KUKA KRL program: f1_Kuka_APT225T02S25.SRC

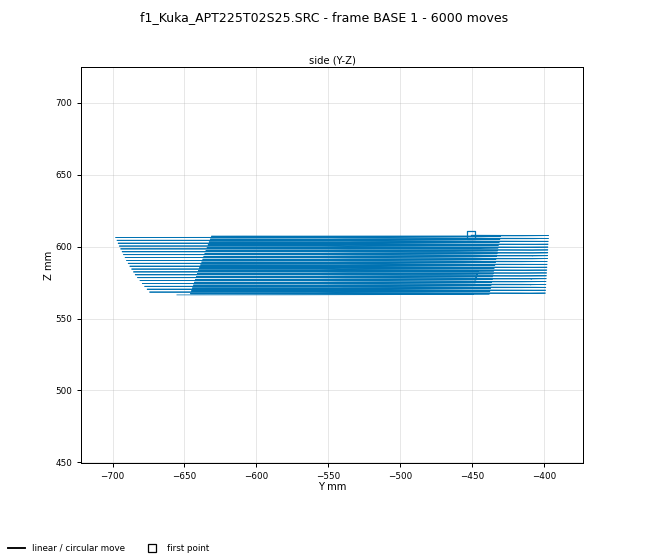
[picture p0: tool path of f1_Kuka_APT225T02S25.SRC in frame BASE 1, 6000 of 6001 moves have a stored position in this frame; points joined in program order, loops and branches not executed]
&ACCESS RVP
&REL 2
&PARAM TEMPLATE = C:\KRC\Roboter\Template\vorgabe
&PARAM EDITMASK = *
DEF f1_Kuka_APT225T02S25()


;FOLD INI;%{PE}%V3.2.0,%MKUKATPBASIS,%CINIT,%VCOMMON,%P
  ;FOLD BAS INI;%{E}%V3.2.0,%MKUKATPBASIS,%CINIT,%VINIT,%P
    GLOBAL INTERRUPT DECL 3 WHEN $STOPMESS==TRUE DO IR_STOPM ( )
    INTERRUPT ON 3
    BAS (#INITMOV,0 )
  ;ENDFOLD (BAS INI)
  ;FOLD USER INI;%{E}%V3.2.0,%MKUKATPUSER,%CINIT,%VINIT,%P
    ;Make your modifications here
  ;ENDFOLD (USER INI)
;ENDFOLD (INI)


;*** Make Null PTP Move
  PTP $pos_act

;*** Auto Load The Correct TOOL Data
  $tool=tool_data[2]

;*** Auto Load The Correct BASE Data
  $base=base_data[1]

  $ADVANCE = 5

;*** Restate Last Velocity
MMPM(30000.0)
SetRPM(8000)
LIN {X -0.035,Y -450.597,Z 607.985,A 0.000,B 0.000,C 90.000,E1 213.214} C_DIS
LIN {X 0.136,Y -446.521,Z 607.972,A 0.000,B 0.000,C 90.000,E1 210.924} C_DIS
LIN {X -0.250,Y -442.434,Z 607.959,A 0.000,B 0.000,C 90.000,E1 208.693} C_DIS
LIN {X 0.124,Y -440.119,Z 607.952,A 0.000,B 0.000,C 90.000,E1 207.334} C_DIS
LIN {X -0.104,Y -437.231,Z 607.943,A 0.000,B 0.000,C 90.000,E1 205.720} C_DIS
LIN {X -0.186,Y -434.380,Z 607.934,A 0.000,B 0.000,C 90.000,E1 204.079} C_DIS
LIN {X 0.098,Y -430.481,Z 607.921,A 0.000,B 0.000,C 90.000,E1 201.716} C_DIS
LIN {X -0.046,Y -427.723,Z 607.911,A 0.000,B 0.000,C 90.000,E1 200.066} C_DIS
LIN {X 0.139,Y -423.997,Z 607.898,A 0.000,B 0.000,C 90.000,E1 197.692} C_DIS
LIN {X -0.165,Y -420.659,Z 607.885,A 0.000,B 0.000,C 90.000,E1 195.371} C_DIS
LIN {X -0.117,Y -418.759,Z 607.878,A 0.000,B 0.000,C 90.000,E1 194.008} C_DIS
LIN {X 0.000,Y -415.623,Z 607.866,A 0.000,B 0.000,C 90.000,E1 191.951} C_DIS
LIN {X 0.069,Y -411.377,Z 607.849,A 0.000,B 0.000,C 90.000,E1 188.859} C_DIS
LIN {X 0.166,Y -409.163,Z 607.840,A 0.000,B 0.000,C 90.000,E1 187.125} C_DIS
LIN {X 0.188,Y -406.047,Z 607.826,A 0.000,B 0.000,C 90.000,E1 184.702} C_DIS
LIN {X -0.104,Y -401.893,Z 607.805,A 0.000,B 0.000,C 90.000,E1 180.917} C_DIS
LIN {X 0.005,Y -399.883,Z 607.791,A 0.000,B 0.000,C 90.000,E1 178.453} C_DIS
LIN {X -0.042,Y -397.946,Z 607.772,A 0.000,B 0.000,C 90.000,E1 174.951} C_DIS
LIN {X 0.089,Y -397.239,Z 607.758,A 0.000,B 0.000,C 90.000,E1 172.470} C_DIS
LIN {X -0.143,Y -396.829,Z 607.745,A 0.000,B 0.000,C 90.000,E1 170.038} C_DIS
LIN {X 0.183,Y -396.837,Z 607.729,A 0.000,B 0.000,C 90.000,E1 167.173} C_DIS
LIN {X -0.078,Y -397.303,Z 607.713,A 0.000,B 0.000,C 90.000,E1 164.393} C_DIS
LIN {X 0.094,Y -397.670,Z 607.705,A 0.000,B 0.000,C 90.000,E1 162.960} C_DIS
LIN {X 0.110,Y -398.325,Z 607.692,A 0.000,B 0.000,C 90.000,E1 160.496} C_DIS
LIN {X -0.123,Y -398.904,Z 607.682,A 0.000,B 0.000,C 90.000,E1 158.773} C_DIS
LIN {X -0.113,Y -399.695,Z 607.670,A 0.000,B 0.000,C 90.000,E1 156.666} C_DIS
LIN {X 0.072,Y -400.529,Z 607.659,A 0.000,B 0.000,C 90.000,E1 154.537} C_DIS
LIN {X 0.076,Y -401.373,Z 607.647,A 0.000,B 0.000,C 90.000,E1 152.436} C_DIS
LIN {X -0.127,Y -402.008,Z 607.637,A 0.000,B 0.000,C 90.000,E1 150.717} C_DIS
LIN {X -0.068,Y -402.708,Z 607.626,A 0.000,B 0.000,C 90.000,E1 148.614} C_DIS
LIN {X 0.077,Y -403.311,Z 607.614,A 0.000,B 0.000,C 90.000,E1 146.501} C_DIS
LIN {X 0.131,Y -403.912,Z 607.602,A 0.000,B 0.000,C 90.000,E1 144.402} C_DIS
LIN {X 0.002,Y -404.655,Z 607.589,A 0.000,B 0.000,C 90.000,E1 141.984} C_DIS
LIN {X -0.068,Y -405.359,Z 607.577,A 0.000,B 0.000,C 90.000,E1 139.908} C_DIS
LIN {X 0.004,Y -405.810,Z 607.568,A 0.000,B 0.000,C 90.000,E1 138.162} C_DIS
LIN {X 0.028,Y -406.293,Z 607.554,A 0.000,B 0.000,C 90.000,E1 135.729} C_DIS
LIN {X 0.215,Y -406.624,Z 607.543,A 0.000,B 0.000,C 90.000,E1 133.623} C_DIS
LIN {X -0.133,Y -406.875,Z 607.535,A 0.000,B 0.000,C 90.000,E1 132.285} C_DIS
LIN {X 0.111,Y -407.271,Z 607.523,A 0.000,B 0.000,C 90.000,E1 130.172} C_DIS
LIN {X 0.085,Y -407.637,Z 607.515,A 0.000,B 0.000,C 90.000,E1 128.705} C_DIS
LIN {X 0.252,Y -415.304,Z 607.500,A 0.000,B 0.000,C 90.000,E1 126.011} C_DIS
LIN {X -0.037,Y -417.748,Z 607.495,A 0.000,B 0.000,C 90.000,E1 125.025} C_DIS
LIN {X 0.201,Y -421.789,Z 607.486,A 0.000,B 0.000,C 90.000,E1 123.372} C_DIS
LIN {X 0.162,Y -421.843,Z 607.486,A 0.000,B 0.000,C 90.000,E1 123.372} C_DIS
LIN {X 0.201,Y -422.819,Z 607.485,A 0.000,B 0.000,C 90.000,E1 123.293} C_DIS
LIN {X -0.069,Y -426.964,Z 607.484,A 0.000,B 0.000,C 90.000,E1 123.086} C_DIS
LIN {X -0.088,Y -450.936,Z 607.477,A 0.000,B 0.000,C 90.000,E1 121.878} C_DIS
LIN {X 0.091,Y -460.950,Z 607.474,A 0.000,B 0.000,C 90.000,E1 121.337} C_DIS
LIN {X 0.206,Y -472.469,Z 607.471,A 0.000,B 0.000,C 90.000,E1 120.669} C_DIS
LIN {X -0.047,Y -482.176,Z 607.467,A 0.000,B 0.000,C 90.000,E1 120.129} C_DIS
LIN {X -0.197,Y -488.571,Z 607.465,A 0.000,B 0.000,C 90.000,E1 119.745} C_DIS
LIN {X 0.182,Y -498.111,Z 607.462,A 0.000,B 0.000,C 90.000,E1 119.077} C_DIS
LIN {X -0.210,Y -504.249,Z 607.459,A 0.000,B 0.000,C 90.000,E1 118.693} C_DIS
LIN {X 0.009,Y -511.965,Z 607.456,A 0.000,B 0.000,C 90.000,E1 118.103} C_DIS
LIN {X 0.049,Y -518.096,Z 607.454,A 0.000,B 0.000,C 90.000,E1 117.641} C_DIS
LIN {X -0.222,Y -527.985,Z 607.449,A 0.000,B 0.000,C 90.000,E1 116.873} C_DIS
LIN {X 0.112,Y -533.671,Z 607.447,A 0.000,B 0.000,C 90.000,E1 116.360} C_DIS
LIN {X 0.246,Y -539.267,Z 607.444,A 0.000,B 0.000,C 90.000,E1 115.848} C_DIS
LIN {X -0.034,Y -544.196,Z 607.441,A 0.000,B 0.000,C 90.000,E1 115.412} C_DIS
LIN {X 0.283,Y -549.010,Z 607.439,A 0.000,B 0.000,C 90.000,E1 114.899} C_DIS
LIN {X 0.037,Y -553.759,Z 607.436,A 0.000,B 0.000,C 90.000,E1 114.387} C_DIS
LIN {X 0.105,Y -558.121,Z 607.432,A 0.000,B 0.000,C 90.000,E1 113.823} C_DIS
LIN {X 0.087,Y -562.823,Z 607.429,A 0.000,B 0.000,C 90.000,E1 113.131} C_DIS
LIN {X -0.203,Y -567.599,Z 607.424,A 0.000,B 0.000,C 90.000,E1 112.333} C_DIS
LIN {X 0.089,Y -571.862,Z 607.419,A 0.000,B 0.000,C 90.000,E1 111.482} C_DIS
LIN {X 0.188,Y -575.169,Z 607.416,A 0.000,B 0.000,C 90.000,E1 110.791} C_DIS
LIN {X 0.107,Y -578.237,Z 607.412,A 0.000,B 0.000,C 90.000,E1 110.120} C_DIS
LIN {X -0.031,Y -581.512,Z 607.407,A 0.000,B 0.000,C 90.000,E1 109.322} C_DIS
LIN {X 0.225,Y -584.590,Z 607.403,A 0.000,B 0.000,C 90.000,E1 108.489} C_DIS
LIN {X 0.144,Y -587.415,Z 607.398,A 0.000,B 0.000,C 90.000,E1 107.692} C_DIS
LIN {X 0.156,Y -590.709,Z 607.392,A 0.000,B 0.000,C 90.000,E1 106.622} C_DIS
LIN {X 0.221,Y -593.690,Z 607.387,A 0.000,B 0.000,C 90.000,E1 105.552} C_DIS
LIN {X 0.184,Y -600.514,Z 607.373,A 0.000,B 0.000,C 90.000,E1 103.175} C_DIS
LIN {X 0.275,Y -605.256,Z 607.365,A 0.000,B 0.000,C 90.000,E1 101.591} C_DIS
LIN {X 0.273,Y -608.432,Z 607.359,A 0.000,B 0.000,C 90.000,E1 100.546} C_DIS
LIN {X 0.064,Y -612.242,Z 607.352,A 0.000,B 0.000,C 90.000,E1 99.265} C_DIS
LIN {X -0.179,Y -615.776,Z 607.344,A 0.000,B 0.000,C 90.000,E1 97.992} C_DIS
LIN {X -0.041,Y -618.497,Z 607.339,A 0.000,B 0.000,C 90.000,E1 96.947} C_DIS
LIN {X 0.055,Y -621.080,Z 607.333,A 0.000,B 0.000,C 90.000,E1 95.910} C_DIS
LIN {X -0.119,Y -623.777,Z 607.326,A 0.000,B 0.000,C 90.000,E1 94.645} C_DIS
LIN {X -0.088,Y -624.817,Z 607.323,A 0.000,B 0.000,C 90.000,E1 94.131} C_DIS
LIN {X -0.203,Y -626.978,Z 607.316,A 0.000,B 0.000,C 90.000,E1 92.865} C_DIS
LIN {X -0.069,Y -628.522,Z 607.310,A 0.000,B 0.000,C 90.000,E1 91.835} C_DIS
LIN {X -0.162,Y -630.042,Z 607.303,A 0.000,B 0.000,C 90.000,E1 90.573} C_DIS
LIN {X -0.072,Y -630.506,Z 607.300,A 0.000,B 0.000,C 90.000,E1 90.057} C_DIS
LIN {X 0.118,Y -631.128,Z 607.295,A 0.000,B 0.000,C 90.000,E1 89.026} C_DIS
LIN {X -0.054,Y -631.303,Z 607.290,A 0.000,B 0.000,C 90.000,E1 88.282} C_DIS
LIN {X -0.112,Y -631.250,Z 607.283,A 0.000,B 0.000,C 90.000,E1 87.020} C_DIS
LIN {X 0.015,Y -631.105,Z 607.281,A 0.000,B 0.000,C 90.000,E1 86.502} C_DIS
LIN {X -0.050,Y -630.373,Z 607.274,A 0.000,B 0.000,C 90.000,E1 85.241} C_DIS
LIN {X 0.201,Y -629.528,Z 607.268,A 0.000,B 0.000,C 90.000,E1 84.204} C_DIS
LIN {X -0.180,Y -628.525,Z 607.262,A 0.000,B 0.000,C 90.000,E1 83.223} C_DIS
LIN {X 0.045,Y -627.114,Z 607.257,A 0.000,B 0.000,C 90.000,E1 82.186} C_DIS
LIN {X 0.123,Y -625.043,Z 607.250,A 0.000,B 0.000,C 90.000,E1 80.905} C_DIS
LIN {X -0.221,Y -623.038,Z 607.244,A 0.000,B 0.000,C 90.000,E1 79.916} C_DIS
LIN {X 0.020,Y -620.933,Z 607.238,A 0.000,B 0.000,C 90.000,E1 78.870} C_DIS
LIN {X 0.218,Y -618.647,Z 607.233,A 0.000,B 0.000,C 90.000,E1 77.825} C_DIS
LIN {X -0.094,Y -616.179,Z 607.227,A 0.000,B 0.000,C 90.000,E1 76.825} C_DIS
LIN {X 0.069,Y -612.828,Z 607.220,A 0.000,B 0.000,C 90.000,E1 75.519} C_DIS
LIN {X 0.181,Y -609.203,Z 607.212,A 0.000,B 0.000,C 90.000,E1 74.212} C_DIS
LIN {X -0.003,Y -606.832,Z 607.208,A 0.000,B 0.000,C 90.000,E1 73.449} C_DIS
LIN {X -0.045,Y -604.265,Z 607.204,A 0.000,B 0.000,C 90.000,E1 72.670} C_DIS
LIN {X 0.075,Y -601.395,Z 607.199,A 0.000,B 0.000,C 90.000,E1 71.873} C_DIS
LIN {X -0.312,Y -597.101,Z 607.194,A 0.000,B 0.000,C 90.000,E1 70.859} C_DIS
LIN {X -0.067,Y -591.722,Z 607.187,A 0.000,B 0.000,C 90.000,E1 69.645} C_DIS
LIN {X 0.203,Y -588.653,Z 607.183,A 0.000,B 0.000,C 90.000,E1 68.954} C_DIS
LIN {X 0.169,Y -584.506,Z 607.179,A 0.000,B 0.000,C 90.000,E1 68.156} C_DIS
LIN {X 0.158,Y -580.904,Z 607.175,A 0.000,B 0.000,C 90.000,E1 67.486} C_DIS
LIN {X 0.260,Y -575.959,Z 607.171,A 0.000,B 0.000,C 90.000,E1 66.666} C_DIS
LIN {X -0.279,Y -572.428,Z 607.168,A 0.000,B 0.000,C 90.000,E1 66.177} C_DIS
LIN {X -0.172,Y -567.537,Z 607.164,A 0.000,B 0.000,C 90.000,E1 65.485} C_DIS
LIN {X -0.018,Y -563.248,Z 607.161,A 0.000,B 0.000,C 90.000,E1 64.921} C_DIS
LIN {X 0.103,Y -558.628,Z 607.158,A 0.000,B 0.000,C 90.000,E1 64.357} C_DIS
LIN {X 0.007,Y -553.569,Z 607.155,A 0.000,B 0.000,C 90.000,E1 63.819} C_DIS
LIN {X 0.279,Y -547.976,Z 607.152,A 0.000,B 0.000,C 90.000,E1 63.256} C_DIS
LIN {X -0.135,Y -543.643,Z 607.150,A 0.000,B 0.000,C 90.000,E1 62.922} C_DIS
LIN {X -0.010,Y -539.017,Z 607.148,A 0.000,B 0.000,C 90.000,E1 62.564} C_DIS
LIN {X 0.105,Y -533.075,Z 607.145,A 0.000,B 0.000,C 90.000,E1 62.153} C_DIS
LIN {X -0.007,Y -526.442,Z 607.143,A 0.000,B 0.000,C 90.000,E1 61.769} C_DIS
LIN {X 0.051,Y -519.547,Z 607.141,A 0.000,B 0.000,C 90.000,E1 61.385} C_DIS
LIN {X 0.000,Y -512.850,Z 607.139,A 0.000,B 0.000,C 90.000,E1 61.051} C_DIS
LIN {X 0.227,Y -500.895,Z 607.136,A 0.000,B 0.000,C 90.000,E1 60.461} C_DIS
LIN {X -0.159,Y -485.528,Z 607.132,A 0.000,B 0.000,C 90.000,E1 59.793} C_DIS
LIN {X -0.080,Y -468.875,Z 607.128,A 0.000,B 0.000,C 90.000,E1 58.997} C_DIS
LIN {X -0.240,Y -446.443,Z 607.121,A 0.000,B 0.000,C 90.000,E1 57.867} C_DIS
LIN {X -0.043,Y -446.380,Z 607.121,A 0.000,B 0.000,C 90.000,E1 57.837} C_DIS
LIN {X -0.065,Y -443.942,Z 607.114,A 0.000,B 0.000,C 90.000,E1 56.501} C_DIS
LIN {X 0.223,Y -434.128,Z 607.090,A 0.000,B 0.000,C 90.000,E1 52.190} C_DIS
LIN {X 0.064,Y -431.651,Z 607.083,A 0.000,B 0.000,C 90.000,E1 50.884} C_DIS
LIN {X -0.013,Y -430.264,Z 607.080,A 0.000,B 0.000,C 90.000,E1 50.312} C_DIS
LIN {X 0.057,Y -431.003,Z 607.074,A 0.000,B 0.000,C 90.000,E1 49.218} C_DIS
LIN {X 0.055,Y -432.039,Z 607.064,A 0.000,B 0.000,C 90.000,E1 47.553} C_DIS
LIN {X -0.083,Y -433.331,Z 607.051,A 0.000,B 0.000,C 90.000,E1 45.243} C_DIS
LIN {X -0.124,Y -434.602,Z 607.040,A 0.000,B 0.000,C 90.000,E1 43.257} C_DIS
LIN {X -0.086,Y -435.484,Z 607.031,A 0.000,B 0.000,C 90.000,E1 41.595} C_DIS
LIN {X 0.055,Y -436.199,Z 607.024,A 0.000,B 0.000,C 90.000,E1 40.253} C_DIS
LIN {X 0.158,Y -437.105,Z 607.013,A 0.000,B 0.000,C 90.000,E1 38.257} C_DIS
LIN {X 0.055,Y -437.585,Z 607.005,A 0.000,B 0.000,C 90.000,E1 36.950} C_DIS
LIN {X 0.005,Y -438.149,Z 606.994,A 0.000,B 0.000,C 90.000,E1 34.978} C_DIS
LIN {X -0.017,Y -438.398,Z 606.989,A 0.000,B 0.000,C 90.000,E1 33.992} C_DIS
LIN {X -0.009,Y -438.614,Z 606.982,A 0.000,B 0.000,C 90.000,E1 32.673} C_DIS
LIN {X -0.131,Y -439.071,Z 606.969,A 0.000,B 0.000,C 90.000,E1 30.384} C_DIS
LIN {X 0.124,Y -439.584,Z 606.954,A 0.000,B 0.000,C 90.000,E1 27.719} C_DIS
LIN {X -0.070,Y -440.005,Z 606.943,A 0.000,B 0.000,C 90.000,E1 25.771} C_DIS
LIN {X 0.001,Y -440.595,Z 606.930,A 0.000,B 0.000,C 90.000,E1 23.462} C_DIS
LIN {X -0.178,Y -441.093,Z 606.921,A 0.000,B 0.000,C 90.000,E1 21.844} C_DIS
LIN {X -0.099,Y -441.754,Z 606.910,A 0.000,B 0.000,C 90.000,E1 19.866} C_DIS
LIN {X -0.182,Y -442.594,Z 606.898,A 0.000,B 0.000,C 90.000,E1 17.583} C_DIS
LIN {X -0.086,Y -443.742,Z 606.883,A 0.000,B 0.000,C 90.000,E1 14.954} C_DIS
LIN {X 0.074,Y -445.001,Z 606.870,A 0.000,B 0.000,C 90.000,E1 12.647} C_DIS
LIN {X -0.014,Y -446.977,Z 606.854,A 0.000,B 0.000,C 90.000,E1 9.726} C_DIS
LIN {X -0.124,Y -448.697,Z 606.841,A 0.000,B 0.000,C 90.000,E1 7.466} C_DIS
LIN {X 0.150,Y -450.682,Z 606.829,A 0.000,B 0.000,C 90.000,E1 5.163} C_DIS
LIN {X -0.195,Y -452.646,Z 606.818,A 0.000,B 0.000,C 90.000,E1 3.269} C_DIS
LIN {X 0.133,Y -455.148,Z 606.806,A 0.000,B 0.000,C 90.000,E1 0.974} C_DIS
LIN {X 0.198,Y -458.826,Z 606.790,A 0.000,B 0.000,C 90.000,E1 358.167} C_DIS
LIN {X 0.211,Y -463.082,Z 606.774,A 0.000,B 0.000,C 90.000,E1 355.298} C_DIS
LIN {X -0.021,Y -466.682,Z 606.762,A 0.000,B 0.000,C 90.000,E1 353.109} C_DIS
LIN {X 0.064,Y -468.724,Z 606.755,A 0.000,B 0.000,C 90.000,E1 351.837} C_DIS
LIN {X -0.184,Y -471.670,Z 606.744,A 0.000,B 0.000,C 90.000,E1 349.982} C_DIS
LIN {X -0.213,Y -476.388,Z 606.729,A 0.000,B 0.000,C 90.000,E1 347.173} C_DIS
LIN {X -0.174,Y -480.851,Z 606.715,A 0.000,B 0.000,C 90.000,E1 344.685} C_DIS
LIN {X 0.132,Y -484.857,Z 606.703,A 0.000,B 0.000,C 90.000,E1 342.489} C_DIS
LIN {X -0.119,Y -488.395,Z 606.693,A 0.000,B 0.000,C 90.000,E1 340.678} C_DIS
LIN {X 0.011,Y -491.298,Z 606.684,A 0.000,B 0.000,C 90.000,E1 339.135} C_DIS
LIN {X 0.022,Y -494.148,Z 606.676,A 0.000,B 0.000,C 90.000,E1 337.614} C_DIS
LIN {X 0.002,Y -496.691,Z 606.667,A 0.000,B 0.000,C 90.000,E1 336.102} C_DIS
LIN {X 0.038,Y -499.097,Z 606.659,A 0.000,B 0.000,C 90.000,E1 334.588} C_DIS
LIN {X 0.109,Y -501.413,Z 606.651,A 0.000,B 0.000,C 90.000,E1 333.076} C_DIS
LIN {X -0.083,Y -504.481,Z 606.639,A 0.000,B 0.000,C 90.000,E1 331.001} C_DIS
LIN {X -0.020,Y -507.133,Z 606.629,A 0.000,B 0.000,C 90.000,E1 329.203} C_DIS
LIN {X 0.041,Y -513.810,Z 606.608,A 0.000,B 0.000,C 90.000,E1 325.341} C_DIS
LIN {X -0.109,Y -518.674,Z 606.594,A 0.000,B 0.000,C 90.000,E1 323.004} C_DIS
LIN {X 0.034,Y -520.601,Z 606.590,A 0.000,B 0.000,C 90.000,E1 322.110} C_DIS
LIN {X -0.121,Y -522.861,Z 606.585,A 0.000,B 0.000,C 90.000,E1 321.251} C_DIS
LIN {X -0.025,Y -524.466,Z 606.582,A 0.000,B 0.000,C 90.000,E1 320.803} C_DIS
LIN {X -0.068,Y -525.798,Z 606.581,A 0.000,B 0.000,C 90.000,E1 320.517} C_DIS
LIN {X -0.214,Y -527.777,Z 606.579,A 0.000,B 0.000,C 90.000,E1 320.194} C_DIS
LIN {X -0.089,Y -531.075,Z 606.576,A 0.000,B 0.000,C 90.000,E1 319.747} C_DIS
LIN {X 0.087,Y -537.928,Z 606.573,A 0.000,B 0.000,C 90.000,E1 319.057} C_DIS
LIN {X 0.247,Y -541.779,Z 606.571,A 0.000,B 0.000,C 90.000,E1 318.690} C_DIS
LIN {X 0.145,Y -552.956,Z 606.566,A 0.000,B 0.000,C 90.000,E1 317.838} C_DIS
LIN {X 0.074,Y -565.994,Z 606.560,A 0.000,B 0.000,C 90.000,E1 316.824} C_DIS
LIN {X 0.158,Y -583.534,Z 606.553,A 0.000,B 0.000,C 90.000,E1 315.486} C_DIS
LIN {X -0.210,Y -589.167,Z 606.550,A 0.000,B 0.000,C 90.000,E1 315.081} C_DIS
LIN {X 0.071,Y -594.707,Z 606.548,A 0.000,B 0.000,C 90.000,E1 314.595} C_DIS
LIN {X 0.000,Y -602.986,Z 606.544,A 0.000,B 0.000,C 90.000,E1 313.905} C_DIS
LIN {X 0.042,Y -609.408,Z 606.541,A 0.000,B 0.000,C 90.000,E1 313.299} C_DIS
LIN {X -0.052,Y -613.115,Z 606.539,A 0.000,B 0.000,C 90.000,E1 312.933} C_DIS
LIN {X 0.000,Y -619.109,Z 606.535,A 0.000,B 0.000,C 90.000,E1 312.285} C_DIS
LIN {X 0.014,Y -625.843,Z 606.531,A 0.000,B 0.000,C 90.000,E1 311.515} C_DIS
LIN {X 0.108,Y -632.154,Z 606.526,A 0.000,B 0.000,C 90.000,E1 310.744} C_DIS
LIN {X 0.227,Y -639.295,Z 606.522,A 0.000,B 0.000,C 90.000,E1 309.850} C_DIS
LIN {X 0.118,Y -642.249,Z 606.519,A 0.000,B 0.000,C 90.000,E1 309.483} C_DIS
LIN {X -0.066,Y -646.944,Z 606.516,A 0.000,B 0.000,C 90.000,E1 308.874} C_DIS
LIN {X 0.370,Y -649.589,Z 606.514,A 0.000,B 0.000,C 90.000,E1 308.463} C_DIS
LIN {X 0.312,Y -652.177,Z 606.512,A 0.000,B 0.000,C 90.000,E1 308.096} C_DIS
LIN {X -0.196,Y -656.043,Z 606.508,A 0.000,B 0.000,C 90.000,E1 307.523} C_DIS
LIN {X -0.188,Y -658.978,Z 606.506,A 0.000,B 0.000,C 90.000,E1 307.030} C_DIS
LIN {X 0.280,Y -662.262,Z 606.502,A 0.000,B 0.000,C 90.000,E1 306.377} C_DIS
LIN {X -0.205,Y -664.698,Z 606.500,A 0.000,B 0.000,C 90.000,E1 305.931} C_DIS
LIN {X -0.026,Y -667.987,Z 606.495,A 0.000,B 0.000,C 90.000,E1 305.185} C_DIS
LIN {X 0.023,Y -671.013,Z 606.491,A 0.000,B 0.000,C 90.000,E1 304.452} C_DIS
LIN {X -0.136,Y -674.742,Z 606.486,A 0.000,B 0.000,C 90.000,E1 303.499} C_DIS
LIN {X -0.068,Y -679.013,Z 606.479,A 0.000,B 0.000,C 90.000,E1 302.291} C_DIS
LIN {X 0.079,Y -683.105,Z 606.473,A 0.000,B 0.000,C 90.000,E1 301.082} C_DIS
LIN {X 0.075,Y -686.296,Z 606.467,A 0.000,B 0.000,C 90.000,E1 300.129} C_DIS
LIN {X 0.219,Y -691.028,Z 606.460,A 0.000,B 0.000,C 90.000,E1 298.693} C_DIS
LIN {X -0.041,Y -693.841,Z 606.454,A 0.000,B 0.000,C 90.000,E1 297.769} C_DIS
LIN {X 0.088,Y -695.800,Z 606.450,A 0.000,B 0.000,C 90.000,E1 297.052} C_DIS
LIN {X -0.338,Y -696.997,Z 606.448,A 0.000,B 0.000,C 90.000,E1 296.616} C_DIS
LIN {X -0.184,Y -697.868,Z 606.444,A 0.000,B 0.000,C 90.000,E1 295.899} C_DIS
LIN {X 0.039,Y -697.209,Z 606.441,A 0.000,B 0.000,C 90.000,E1 295.412} C_DIS
LIN {X 0.301,Y -696.791,Z 606.440,A 0.000,B 0.000,C 90.000,E1 295.155} C_DIS
LIN {X -0.199,Y -696.311,Z 606.439,A 0.000,B 0.000,C 90.000,E1 295.079} C_DIS
LIN {X 0.146,Y -692.274,Z 606.436,A 0.000,B 0.000,C 90.000,E1 294.463} C_DIS
LIN {X 0.268,Y -690.959,Z 606.435,A 0.000,B 0.000,C 90.000,E1 294.335} C_DIS
LIN {X -0.151,Y -685.572,Z 606.434,A 0.000,B 0.000,C 90.000,E1 294.079} C_DIS
LIN {X 0.189,Y -682.228,Z 606.433,A 0.000,B 0.000,C 90.000,E1 293.898} C_DIS
LIN {X -0.003,Y -677.283,Z 606.432,A 0.000,B 0.000,C 90.000,E1 293.770} C_DIS
LIN {X -0.103,Y -673.674,Z 606.432,A 0.000,B 0.000,C 90.000,E1 293.695} C_DIS
LIN {X -0.121,Y -661.564,Z 606.431,A 0.000,B 0.000,C 90.000,E1 293.515} C_DIS
LIN {X -0.302,Y -650.735,Z 606.430,A 0.000,B 0.000,C 90.000,E1 293.387} C_DIS
LIN {X 0.024,Y -637.633,Z 606.429,A 0.000,B 0.000,C 90.000,E1 293.131} C_DIS
LIN {X -0.237,Y -628.137,Z 606.427,A 0.000,B 0.000,C 90.000,E1 292.950} C_DIS
LIN {X 0.344,Y -618.349,Z 606.426,A 0.000,B 0.000,C 90.000,E1 292.642} C_DIS
LIN {X -0.062,Y -591.007,Z 606.421,A 0.000,B 0.000,C 90.000,E1 291.844} C_DIS
LIN {X -0.116,Y -578.793,Z 606.419,A 0.000,B 0.000,C 90.000,E1 291.461} C_DIS
LIN {X -0.310,Y -569.980,Z 606.418,A 0.000,B 0.000,C 90.000,E1 291.227} C_DIS
LIN {X -0.041,Y -565.276,Z 606.417,A 0.000,B 0.000,C 90.000,E1 291.046} C_DIS
LIN {X -0.045,Y -560.119,Z 606.416,A 0.000,B 0.000,C 90.000,E1 290.791} C_DIS
LIN {X -0.091,Y -560.055,Z 606.416,A 0.000,B 0.000,C 90.000,E1 290.791} C_DIS
LIN {X -0.155,Y -558.553,Z 606.414,A 0.000,B 0.000,C 90.000,E1 290.610} C_DIS
LIN {X -0.197,Y -558.534,Z 606.414,A 0.000,B 0.000,C 90.000,E1 290.610} C_DIS
LIN {X -0.121,Y -558.032,Z 606.413,A 0.000,B 0.000,C 90.000,E1 290.355} C_DIS
LIN {X -0.076,Y -557.803,Z 606.410,A 0.000,B 0.000,C 90.000,E1 289.758} C_DIS
LIN {X -0.010,Y -557.869,Z 606.402,A 0.000,B 0.000,C 90.000,E1 288.362} C_DIS
LIN {X -0.243,Y -557.663,Z 606.396,A 0.000,B 0.000,C 90.000,E1 287.275} C_DIS
LIN {X 0.048,Y -557.359,Z 606.390,A 0.000,B 0.000,C 90.000,E1 286.134} C_DIS
LIN {X 0.050,Y -557.001,Z 606.385,A 0.000,B 0.000,C 90.000,E1 285.300} C_DIS
LIN {X -0.102,Y -556.202,Z 606.376,A 0.000,B 0.000,C 90.000,E1 283.647} C_DIS
LIN {X 0.151,Y -555.323,Z 606.367,A 0.000,B 0.000,C 90.000,E1 281.951} C_DIS
LIN {X -0.031,Y -554.322,Z 606.356,A 0.000,B 0.000,C 90.000,E1 280.018} C_DIS
LIN {X 0.113,Y -553.278,Z 606.345,A 0.000,B 0.000,C 90.000,E1 278.049} C_DIS
LIN {X -0.227,Y -552.158,Z 606.331,A 0.000,B 0.000,C 90.000,E1 275.568} C_DIS
LIN {X 0.235,Y -551.526,Z 606.322,A 0.000,B 0.000,C 90.000,E1 273.841} C_DIS
LIN {X 0.118,Y -550.982,Z 606.311,A 0.000,B 0.000,C 90.000,E1 271.892} C_DIS
LIN {X -0.123,Y -550.606,Z 606.303,A 0.000,B 0.000,C 90.000,E1 270.516} C_DIS
LIN {X 0.110,Y -550.267,Z 606.297,A 0.000,B 0.000,C 90.000,E1 269.370} C_DIS
LIN {X -0.091,Y -549.627,Z 606.287,A 0.000,B 0.000,C 90.000,E1 267.707} C_DIS
LIN {X 0.237,Y -548.887,Z 606.278,A 0.000,B 0.000,C 90.000,E1 265.988} C_DIS
LIN {X -0.014,Y -548.148,Z 606.270,A 0.000,B 0.000,C 90.000,E1 264.609} C_DIS
LIN {X -0.221,Y -547.272,Z 606.262,A 0.000,B 0.000,C 90.000,E1 263.223} C_DIS
LIN {X 0.085,Y -546.303,Z 606.256,A 0.000,B 0.000,C 90.000,E1 262.064} C_DIS
LIN {X -0.154,Y -545.035,Z 606.248,A 0.000,B 0.000,C 90.000,E1 260.679} C_DIS
LIN {X -0.166,Y -543.109,Z 606.237,A 0.000,B 0.000,C 90.000,E1 258.701} C_DIS
LIN {X -0.165,Y -541.794,Z 606.229,A 0.000,B 0.000,C 90.000,E1 257.285} C_DIS
LIN {X -0.306,Y -540.422,Z 606.221,A 0.000,B 0.000,C 90.000,E1 255.880} C_DIS
LIN {X -0.208,Y -538.982,Z 606.214,A 0.000,B 0.000,C 90.000,E1 254.448} C_DIS
LIN {X -0.128,Y -537.515,Z 606.206,A 0.000,B 0.000,C 90.000,E1 253.015} C_DIS
LIN {X -0.084,Y -536.051,Z 606.198,A 0.000,B 0.000,C 90.000,E1 251.583} C_DIS
LIN {X 0.066,Y -534.770,Z 606.191,A 0.000,B 0.000,C 90.000,E1 250.423} C_DIS
LIN {X 0.199,Y -533.081,Z 606.185,A 0.000,B 0.000,C 90.000,E1 249.263} C_DIS
LIN {X 0.108,Y -531.674,Z 606.180,A 0.000,B 0.000,C 90.000,E1 248.411} C_DIS
LIN {X -0.102,Y -529.680,Z 606.174,A 0.000,B 0.000,C 90.000,E1 247.283} C_DIS
LIN {X -0.152,Y -526.977,Z 606.166,A 0.000,B 0.000,C 90.000,E1 245.845} C_DIS
LIN {X 0.053,Y -524.604,Z 606.159,A 0.000,B 0.000,C 90.000,E1 244.665} C_DIS
LIN {X 0.116,Y -521.501,Z 606.151,A 0.000,B 0.000,C 90.000,E1 243.204} C_DIS
LIN {X 0.223,Y -518.844,Z 606.145,A 0.000,B 0.000,C 90.000,E1 242.025} C_DIS
LIN {X -0.067,Y -516.795,Z 606.140,A 0.000,B 0.000,C 90.000,E1 241.179} C_DIS
LIN {X -0.017,Y -512.514,Z 606.130,A 0.000,B 0.000,C 90.000,E1 239.410} C_DIS
LIN {X 0.124,Y -508.973,Z 606.122,A 0.000,B 0.000,C 90.000,E1 237.916} C_DIS
LIN {X -0.118,Y -505.880,Z 606.115,A 0.000,B 0.000,C 90.000,E1 236.755} C_DIS
LIN {X 0.010,Y -502.586,Z 606.109,A 0.000,B 0.000,C 90.000,E1 235.548} C_DIS
LIN {X 0.265,Y -496.783,Z 606.097,A 0.000,B 0.000,C 90.000,E1 233.417} C_DIS
LIN {X 0.126,Y -492.094,Z 606.087,A 0.000,B 0.000,C 90.000,E1 231.618} C_DIS
LIN {X -0.179,Y -488.936,Z 606.080,A 0.000,B 0.000,C 90.000,E1 230.436} C_DIS
LIN {X 0.155,Y -485.833,Z 606.073,A 0.000,B 0.000,C 90.000,E1 229.175} C_DIS
LIN {X -0.218,Y -480.412,Z 606.061,A 0.000,B 0.000,C 90.000,E1 227.067} C_DIS
LIN {X 0.171,Y -475.861,Z 606.051,A 0.000,B 0.000,C 90.000,E1 225.162} C_DIS
LIN {X 0.110,Y -471.467,Z 606.041,A 0.000,B 0.000,C 90.000,E1 223.299} C_DIS
LIN {X -0.186,Y -468.683,Z 606.034,A 0.000,B 0.000,C 90.000,E1 222.081} C_DIS
LIN {X -0.234,Y -463.076,Z 606.020,A 0.000,B 0.000,C 90.000,E1 219.564} C_DIS
LIN {X -0.166,Y -459.116,Z 606.009,A 0.000,B 0.000,C 90.000,E1 217.649} C_DIS
LIN {X -0.010,Y -454.675,Z 605.997,A 0.000,B 0.000,C 90.000,E1 215.391} C_DIS
LIN {X -0.229,Y -450.352,Z 605.984,A 0.000,B 0.000,C 90.000,E1 213.166} C_DIS
LIN {X -0.200,Y -447.412,Z 605.975,A 0.000,B 0.000,C 90.000,E1 211.544} C_DIS
LIN {X 0.017,Y -445.686,Z 605.970,A 0.000,B 0.000,C 90.000,E1 210.541} C_DIS
LIN {X 0.165,Y -442.185,Z 605.959,A 0.000,B 0.000,C 90.000,E1 208.565} C_DIS
LIN {X -0.018,Y -439.280,Z 605.950,A 0.000,B 0.000,C 90.000,E1 206.950} C_DIS
LIN {X -0.095,Y -436.989,Z 605.942,A 0.000,B 0.000,C 90.000,E1 205.643} C_DIS
LIN {X 0.207,Y -434.153,Z 605.933,A 0.000,B 0.000,C 90.000,E1 203.951} C_DIS
LIN {X -0.078,Y -430.274,Z 605.920,A 0.000,B 0.000,C 90.000,E1 201.663} C_DIS
LIN {X 0.128,Y -426.973,Z 605.909,A 0.000,B 0.000,C 90.000,E1 199.631} C_DIS
LIN {X 0.152,Y -423.332,Z 605.896,A 0.000,B 0.000,C 90.000,E1 197.275} C_DIS
LIN {X 0.179,Y -420.503,Z 605.885,A 0.000,B 0.000,C 90.000,E1 195.245} C_DIS
LIN {X 0.219,Y -418.612,Z 605.877,A 0.000,B 0.000,C 90.000,E1 193.883} C_DIS
LIN {X -0.084,Y -415.498,Z 605.866,A 0.000,B 0.000,C 90.000,E1 191.883} C_DIS
LIN {X -0.098,Y -411.255,Z 605.849,A 0.000,B 0.000,C 90.000,E1 188.803} C_DIS
LIN {X 0.025,Y -409.537,Z 605.841,A 0.000,B 0.000,C 90.000,E1 187.409} C_DIS
LIN {X 0.015,Y -406.402,Z 605.828,A 0.000,B 0.000,C 90.000,E1 184.992} C_DIS
LIN {X 0.131,Y -401.882,Z 605.805,A 0.000,B 0.000,C 90.000,E1 180.802} C_DIS
LIN {X 0.204,Y -399.645,Z 605.789,A 0.000,B 0.000,C 90.000,E1 177.993} C_DIS
LIN {X 0.190,Y -398.010,Z 605.772,A 0.000,B 0.000,C 90.000,E1 174.837} C_DIS
LIN {X -0.051,Y -397.397,Z 605.760,A 0.000,B 0.000,C 90.000,E1 172.761} C_DIS
LIN {X 0.082,Y -396.912,Z 605.744,A 0.000,B 0.000,C 90.000,E1 169.926} C_DIS
LIN {X 0.018,Y -396.964,Z 605.729,A 0.000,B 0.000,C 90.000,E1 167.117} C_DIS
LIN {X -0.104,Y -397.648,Z 605.709,A 0.000,B 0.000,C 90.000,E1 163.614} C_DIS
LIN {X -0.079,Y -398.303,Z 605.695,A 0.000,B 0.000,C 90.000,E1 161.148} C_DIS
LIN {X 0.004,Y -398.979,Z 605.684,A 0.000,B 0.000,C 90.000,E1 159.028} C_DIS
LIN {X 0.083,Y -399.891,Z 605.670,A 0.000,B 0.000,C 90.000,E1 156.561} C_DIS
LIN {X -0.041,Y -400.457,Z 605.662,A 0.000,B 0.000,C 90.000,E1 155.177} C_DIS
LIN {X -0.156,Y -401.488,Z 605.648,A 0.000,B 0.000,C 90.000,E1 152.743} C_DIS
LIN {X 0.002,Y -402.119,Z 605.639,A 0.000,B 0.000,C 90.000,E1 150.973} C_DIS
LIN {X 0.069,Y -402.836,Z 605.627,A 0.000,B 0.000,C 90.000,E1 148.869} C_DIS
LIN {X 0.210,Y -403.249,Z 605.619,A 0.000,B 0.000,C 90.000,E1 147.454} C_DIS
LIN {X 0.035,Y -403.851,Z 605.608,A 0.000,B 0.000,C 90.000,E1 145.388} C_DIS
LIN {X 0.208,Y -404.320,Z 605.598,A 0.000,B 0.000,C 90.000,E1 143.623} C_DIS
LIN {X 0.201,Y -405.008,Z 605.587,A 0.000,B 0.000,C 90.000,E1 141.537} C_DIS
LIN {X -0.134,Y -405.463,Z 605.579,A 0.000,B 0.000,C 90.000,E1 140.194} C_DIS
LIN {X -0.057,Y -405.929,Z 605.569,A 0.000,B 0.000,C 90.000,E1 138.447} C_DIS
LIN {X 0.272,Y -406.411,Z 605.556,A 0.000,B 0.000,C 90.000,E1 135.972} C_DIS
LIN {X -0.114,Y -406.718,Z 605.544,A 0.000,B 0.000,C 90.000,E1 133.947} C_DIS
LIN {X -0.046,Y -406.998,Z 605.534,A 0.000,B 0.000,C 90.000,E1 132.204} C_DIS
LIN {X 0.200,Y -407.350,Z 605.523,A 0.000,B 0.000,C 90.000,E1 130.092} C_DIS
LIN {X -0.101,Y -407.644,Z 605.515,A 0.000,B 0.000,C 90.000,E1 128.749} C_DIS
LIN {X -0.071,Y -411.392,Z 605.508,A 0.000,B 0.000,C 90.000,E1 127.363} C_DIS
LIN {X 0.101,Y -415.511,Z 605.500,A 0.000,B 0.000,C 90.000,E1 125.964} C_DIS
LIN {X 0.103,Y -422.582,Z 605.484,A 0.000,B 0.000,C 90.000,E1 123.086} C_DIS
LIN {X 0.064,Y -422.600,Z 605.484,A 0.000,B 0.000,C 90.000,E1 123.086} C_DIS
LIN {X -0.119,Y -427.455,Z 605.482,A 0.000,B 0.000,C 90.000,E1 122.832} C_DIS
LIN {X -0.195,Y -448.349,Z 605.477,A 0.000,B 0.000,C 90.000,E1 121.799} C_DIS
LIN {X -0.043,Y -460.205,Z 605.473,A 0.000,B 0.000,C 90.000,E1 121.180} C_DIS
LIN {X -0.280,Y -469.921,Z 605.470,A 0.000,B 0.000,C 90.000,E1 120.669} C_DIS
LIN {X -0.071,Y -479.817,Z 605.467,A 0.000,B 0.000,C 90.000,E1 120.079} C_DIS
LIN {X -0.007,Y -487.649,Z 605.464,A 0.000,B 0.000,C 90.000,E1 119.589} C_DIS
LIN {X 0.264,Y -497.130,Z 605.461,A 0.000,B 0.000,C 90.000,E1 118.949} C_DIS
LIN {X 0.001,Y -503.198,Z 605.459,A 0.000,B 0.000,C 90.000,E1 118.565} C_DIS
LIN {X 0.214,Y -509.335,Z 605.456,A 0.000,B 0.000,C 90.000,E1 118.103} C_DIS
LIN {X 0.025,Y -518.276,Z 605.453,A 0.000,B 0.000,C 90.000,E1 117.462} C_DIS
LIN {X 0.256,Y -528.559,Z 605.448,A 0.000,B 0.000,C 90.000,E1 116.616} C_DIS
LIN {X 0.071,Y -534.309,Z 605.445,A 0.000,B 0.000,C 90.000,E1 116.155} C_DIS
LIN {X 0.017,Y -539.924,Z 605.443,A 0.000,B 0.000,C 90.000,E1 115.668} C_DIS
LIN {X 0.048,Y -544.037,Z 605.441,A 0.000,B 0.000,C 90.000,E1 115.283} C_DIS
LIN {X 0.010,Y -548.041,Z 605.438,A 0.000,B 0.000,C 90.000,E1 114.899} C_DIS
LIN {X 0.244,Y -552.970,Z 605.435,A 0.000,B 0.000,C 90.000,E1 114.335} C_DIS
LIN {X 0.030,Y -557.249,Z 605.432,A 0.000,B 0.000,C 90.000,E1 113.823} C_DIS
LIN {X -0.167,Y -559.959,Z 605.430,A 0.000,B 0.000,C 90.000,E1 113.462} C_DIS
LIN {X 0.033,Y -562.884,Z 605.428,A 0.000,B 0.000,C 90.000,E1 113.025} C_DIS
LIN {X -0.156,Y -566.851,Z 605.424,A 0.000,B 0.000,C 90.000,E1 112.386} C_DIS
LIN {X 0.123,Y -571.271,Z 605.420,A 0.000,B 0.000,C 90.000,E1 111.535} C_DIS
LIN {X -0.075,Y -575.315,Z 605.415,A 0.000,B 0.000,C 90.000,E1 110.737} C_DIS
LIN {X -0.154,Y -578.428,Z 605.411,A 0.000,B 0.000,C 90.000,E1 110.066} C_DIS
LIN {X -0.289,Y -581.773,Z 605.407,A 0.000,B 0.000,C 90.000,E1 109.268} C_DIS
LIN {X 0.156,Y -584.882,Z 605.402,A 0.000,B 0.000,C 90.000,E1 108.417} C_DIS
LIN {X -0.105,Y -587.737,Z 605.398,A 0.000,B 0.000,C 90.000,E1 107.638} C_DIS
LIN {X -0.017,Y -589.470,Z 605.395,A 0.000,B 0.000,C 90.000,E1 107.094} C_DIS
LIN {X -0.232,Y -591.877,Z 605.391,A 0.000,B 0.000,C 90.000,E1 106.315} C_DIS
LIN {X 0.116,Y -595.567,Z 605.383,A 0.000,B 0.000,C 90.000,E1 104.954} C_DIS
LIN {X -0.034,Y -601.061,Z 605.373,A 0.000,B 0.000,C 90.000,E1 103.119} C_DIS
LIN {X -0.248,Y -605.097,Z 605.366,A 0.000,B 0.000,C 90.000,E1 101.827} C_DIS
LIN {X 0.080,Y -609.104,Z 605.358,A 0.000,B 0.000,C 90.000,E1 100.489} C_DIS
LIN {X 0.140,Y -612.222,Z 605.353,A 0.000,B 0.000,C 90.000,E1 99.443} C_DIS
LIN {X -0.009,Y -615.836,Z 605.345,A 0.000,B 0.000,C 90.000,E1 98.163} C_DIS
LIN {X -0.197,Y -619.279,Z 605.338,A 0.000,B 0.000,C 90.000,E1 96.891} C_DIS
LIN {X -0.090,Y -621.878,Z 605.333,A 0.000,B 0.000,C 90.000,E1 95.853} C_DIS
LIN {X -0.251,Y -624.616,Z 605.325,A 0.000,B 0.000,C 90.000,E1 94.588} C_DIS
LIN {X -0.214,Y -625.637,Z 605.323,A 0.000,B 0.000,C 90.000,E1 94.073} C_DIS
LIN {X 0.313,Y -627.821,Z 605.315,A 0.000,B 0.000,C 90.000,E1 92.751} C_DIS
LIN {X -0.148,Y -629.350,Z 605.310,A 0.000,B 0.000,C 90.000,E1 91.776} C_DIS
LIN {X 0.292,Y -630.322,Z 605.306,A 0.000,B 0.000,C 90.000,E1 90.974} C_DIS
LIN {X 0.116,Y -631.101,Z 605.301,A 0.000,B 0.000,C 90.000,E1 90.229} C_DIS
LIN {X 0.049,Y -631.913,Z 605.294,A 0.000,B 0.000,C 90.000,E1 88.969} C_DIS
LIN {X 0.271,Y -632.090,Z 605.289,A 0.000,B 0.000,C 90.000,E1 87.936} C_DIS
LIN {X 0.238,Y -631.928,Z 605.282,A 0.000,B 0.000,C 90.000,E1 86.674} C_DIS
LIN {X 0.191,Y -631.184,Z 605.275,A 0.000,B 0.000,C 90.000,E1 85.412} C_DIS
LIN {X 0.045,Y -630.610,Z 605.270,A 0.000,B 0.000,C 90.000,E1 84.666} C_DIS
LIN {X 0.301,Y -629.640,Z 605.265,A 0.000,B 0.000,C 90.000,E1 83.628} C_DIS
LIN {X 0.211,Y -628.733,Z 605.261,A 0.000,B 0.000,C 90.000,E1 82.875} C_DIS
LIN {X 0.032,Y -627.642,Z 605.256,A 0.000,B 0.000,C 90.000,E1 82.129} C_DIS
LIN {X 0.116,Y -625.462,Z 605.249,A 0.000,B 0.000,C 90.000,E1 80.849} C_DIS
LIN {X -0.009,Y -623.967,Z 605.245,A 0.000,B 0.000,C 90.000,E1 80.095} C_DIS
LIN {X 0.020,Y -621.255,Z 605.238,A 0.000,B 0.000,C 90.000,E1 78.814} C_DIS
LIN {X 0.351,Y -618.915,Z 605.232,A 0.000,B 0.000,C 90.000,E1 77.757} C_DIS
LIN {X 0.050,Y -616.424,Z 605.227,A 0.000,B 0.000,C 90.000,E1 76.756} C_DIS
LIN {X 0.072,Y -613.008,Z 605.219,A 0.000,B 0.000,C 90.000,E1 75.463} C_DIS
LIN {X 0.184,Y -609.303,Z 605.212,A 0.000,B 0.000,C 90.000,E1 74.157} C_DIS
LIN {X 0.171,Y -606.831,Z 605.208,A 0.000,B 0.000,C 90.000,E1 73.378} C_DIS
LIN {X 0.134,Y -604.149,Z 605.203,A 0.000,B 0.000,C 90.000,E1 72.598} C_DIS
LIN {X 0.070,Y -601.177,Z 605.199,A 0.000,B 0.000,C 90.000,E1 71.819} C_DIS
LIN {X -0.028,Y -597.895,Z 605.195,A 0.000,B 0.000,C 90.000,E1 71.040} C_DIS
LIN {X 0.035,Y -594.289,Z 605.190,A 0.000,B 0.000,C 90.000,E1 70.242} C_DIS
LIN {X 0.064,Y -590.580,Z 605.186,A 0.000,B 0.000,C 90.000,E1 69.444} C_DIS
LIN {X 0.172,Y -588.045,Z 605.183,A 0.000,B 0.000,C 90.000,E1 68.901} C_DIS
LIN {X 0.192,Y -584.535,Z 605.179,A 0.000,B 0.000,C 90.000,E1 68.230} C_DIS
LIN {X -0.316,Y -580.049,Z 605.175,A 0.000,B 0.000,C 90.000,E1 67.486} C_DIS
LIN {X -0.044,Y -575.902,Z 605.171,A 0.000,B 0.000,C 90.000,E1 66.794} C_DIS
LIN {X 0.143,Y -571.473,Z 605.167,A 0.000,B 0.000,C 90.000,E1 66.125} C_DIS
LIN {X 0.205,Y -567.802,Z 605.165,A 0.000,B 0.000,C 90.000,E1 65.613} C_DIS
LIN {X -0.243,Y -562.298,Z 605.161,A 0.000,B 0.000,C 90.000,E1 64.973} C_DIS
LIN {X -0.126,Y -557.531,Z 605.158,A 0.000,B 0.000,C 90.000,E1 64.409} C_DIS
LIN {X 0.106,Y -553.655,Z 605.156,A 0.000,B 0.000,C 90.000,E1 63.973} C_DIS
LIN {X -0.022,Y -548.149,Z 605.153,A 0.000,B 0.000,C 90.000,E1 63.461} C_DIS
LIN {X -0.301,Y -542.232,Z 605.150,A 0.000,B 0.000,C 90.000,E1 62.999} C_DIS
LIN {X 0.139,Y -537.533,Z 605.148,A 0.000,B 0.000,C 90.000,E1 62.615} C_DIS
LIN {X 0.038,Y -531.236,Z 605.146,A 0.000,B 0.000,C 90.000,E1 62.231} C_DIS
LIN {X 0.221,Y -521.125,Z 605.143,A 0.000,B 0.000,C 90.000,E1 61.641} C_DIS
LIN {X 0.055,Y -514.305,Z 605.141,A 0.000,B 0.000,C 90.000,E1 61.307} C_DIS
LIN {X 0.200,Y -502.151,Z 605.138,A 0.000,B 0.000,C 90.000,E1 60.717} C_DIS
LIN {X 0.053,Y -485.052,Z 605.133,A 0.000,B 0.000,C 90.000,E1 59.950} C_DIS
LIN {X 0.231,Y -476.667,Z 605.131,A 0.000,B 0.000,C 90.000,E1 59.537} C_DIS
LIN {X 0.158,Y -460.124,Z 605.127,A 0.000,B 0.000,C 90.000,E1 58.742} C_DIS
LIN {X -0.023,Y -446.882,Z 605.123,A 0.000,B 0.000,C 90.000,E1 58.074} C_DIS
LIN {X -0.065,Y -446.834,Z 605.123,A 0.000,B 0.000,C 90.000,E1 58.074} C_DIS
LIN {X -0.028,Y -444.176,Z 605.115,A 0.000,B 0.000,C 90.000,E1 56.628} C_DIS
LIN {X 0.086,Y -442.611,Z 605.111,A 0.000,B 0.000,C 90.000,E1 55.960} C_DIS
LIN {X -0.054,Y -433.742,Z 605.089,A 0.000,B 0.000,C 90.000,E1 52.029} C_DIS
LIN {X -0.213,Y -431.218,Z 605.082,A 0.000,B 0.000,C 90.000,E1 50.723} C_DIS
LIN {X 0.004,Y -430.667,Z 605.081,A 0.000,B 0.000,C 90.000,E1 50.481} C_DIS
LIN {X -0.036,Y -430.663,Z 605.080,A 0.000,B 0.000,C 90.000,E1 50.481} C_DIS
LIN {X 0.111,Y -431.673,Z 605.072,A 0.000,B 0.000,C 90.000,E1 49.013} C_DIS
LIN {X -0.203,Y -432.740,Z 605.063,A 0.000,B 0.000,C 90.000,E1 47.391} C_DIS
LIN {X -0.013,Y -434.123,Z 605.050,A 0.000,B 0.000,C 90.000,E1 45.040} C_DIS
LIN {X -0.046,Y -435.427,Z 605.039,A 0.000,B 0.000,C 90.000,E1 43.056} C_DIS
LIN {X 0.035,Y -436.323,Z 605.030,A 0.000,B 0.000,C 90.000,E1 41.391} C_DIS
LIN {X -0.139,Y -437.006,Z 605.023,A 0.000,B 0.000,C 90.000,E1 40.092} C_DIS
LIN {X -0.023,Y -437.872,Z 605.012,A 0.000,B 0.000,C 90.000,E1 38.096} C_DIS
LIN {X 0.213,Y -438.238,Z 605.006,A 0.000,B 0.000,C 90.000,E1 37.076} C_DIS
LIN {X 0.173,Y -438.778,Z 604.995,A 0.000,B 0.000,C 90.000,E1 35.105} C_DIS
LIN {X 0.190,Y -439.036,Z 604.988,A 0.000,B 0.000,C 90.000,E1 33.785} C_DIS
LIN {X -0.066,Y -439.220,Z 604.982,A 0.000,B 0.000,C 90.000,E1 32.832} C_DIS
LIN {X -0.161,Y -439.606,Z 604.970,A 0.000,B 0.000,C 90.000,E1 30.541} C_DIS
LIN {X -0.095,Y -439.983,Z 604.957,A 0.000,B 0.000,C 90.000,E1 28.231} C_DIS
LIN {X 0.243,Y -440.266,Z 604.950,A 0.000,B 0.000,C 90.000,E1 26.873} C_DIS
LIN {X -0.136,Y -440.659,Z 604.939,A 0.000,B 0.000,C 90.000,E1 24.951} C_DIS
LIN {X 0.106,Y -441.187,Z 604.928,A 0.000,B 0.000,C 90.000,E1 22.950} C_DIS
LIN {X -0.072,Y -441.645,Z 604.919,A 0.000,B 0.000,C 90.000,E1 21.334} C_DIS
LIN {X 0.007,Y -442.185,Z 604.909,A 0.000,B 0.000,C 90.000,E1 19.685} C_DIS
LIN {X 0.222,Y -442.867,Z 604.898,A 0.000,B 0.000,C 90.000,E1 17.692} C_DIS
LIN {X 0.043,Y -444.141,Z 604.882,A 0.000,B 0.000,C 90.000,E1 14.773} C_DIS
LIN {X -0.057,Y -445.187,Z 604.871,A 0.000,B 0.000,C 90.000,E1 12.827} C_DIS
LIN {X 0.052,Y -447.337,Z 604.853,A 0.000,B 0.000,C 90.000,E1 9.557} C_DIS
LIN {X -0.230,Y -448.794,Z 604.842,A 0.000,B 0.000,C 90.000,E1 7.644} C_DIS
LIN {X -0.200,Y -451.041,Z 604.828,A 0.000,B 0.000,C 90.000,E1 5.049} C_DIS
LIN {X -0.059,Y -452.994,Z 604.817,A 0.000,B 0.000,C 90.000,E1 3.094} C_DIS
LIN {X -0.200,Y -455.499,Z 604.805,A 0.000,B 0.000,C 90.000,E1 0.859} C_DIS
LIN {X 0.201,Y -458.981,Z 604.790,A 0.000,B 0.000,C 90.000,E1 358.167} C_DIS
LIN {X 0.219,Y -463.207,Z 604.774,A 0.000,B 0.000,C 90.000,E1 355.298} C_DIS
LIN {X -0.009,Y -466.777,Z 604.762,A 0.000,B 0.000,C 90.000,E1 353.109} C_DIS
LIN {X 0.076,Y -468.788,Z 604.755,A 0.000,B 0.000,C 90.000,E1 351.837} C_DIS
LIN {X -0.169,Y -471.731,Z 604.744,A 0.000,B 0.000,C 90.000,E1 349.982} C_DIS
LIN {X -0.197,Y -476.449,Z 604.729,A 0.000,B 0.000,C 90.000,E1 347.173} C_DIS
LIN {X -0.130,Y -480.308,Z 604.717,A 0.000,B 0.000,C 90.000,E1 344.991} C_DIS
LIN {X -0.016,Y -483.172,Z 604.708,A 0.000,B 0.000,C 90.000,E1 343.433} C_DIS
LIN {X 0.018,Y -486.639,Z 604.698,A 0.000,B 0.000,C 90.000,E1 341.583} C_DIS
LIN {X -0.055,Y -489.634,Z 604.689,A 0.000,B 0.000,C 90.000,E1 340.061} C_DIS
LIN {X 0.003,Y -493.641,Z 604.677,A 0.000,B 0.000,C 90.000,E1 337.922} C_DIS
LIN {X 0.134,Y -495.228,Z 604.672,A 0.000,B 0.000,C 90.000,E1 336.997} C_DIS
LIN {X 0.133,Y -497.715,Z 604.664,A 0.000,B 0.000,C 90.000,E1 335.485} C_DIS
LIN {X -0.269,Y -500.064,Z 604.656,A 0.000,B 0.000,C 90.000,E1 334.024} C_DIS
LIN {X -0.022,Y -501.921,Z 604.649,A 0.000,B 0.000,C 90.000,E1 332.794} C_DIS
LIN {X -0.057,Y -504.538,Z 604.639,A 0.000,B 0.000,C 90.000,E1 331.001} C_DIS
LIN {X -0.104,Y -507.655,Z 604.627,A 0.000,B 0.000,C 90.000,E1 328.918} C_DIS
LIN {X -0.268,Y -513.259,Z 604.609,A 0.000,B 0.000,C 90.000,E1 325.674} C_DIS
LIN {X -0.013,Y -517.959,Z 604.596,A 0.000,B 0.000,C 90.000,E1 323.290} C_DIS
LIN {X -0.040,Y -521.762,Z 604.586,A 0.000,B 0.000,C 90.000,E1 321.537} C_DIS
LIN {X -0.139,Y -523.367,Z 604.583,A 0.000,B 0.000,C 90.000,E1 320.964} C_DIS
LIN {X 0.105,Y -525.762,Z 604.580,A 0.000,B 0.000,C 90.000,E1 320.356} C_DIS
LIN {X -0.083,Y -526.234,Z 604.579,A 0.000,B 0.000,C 90.000,E1 320.231} C_DIS
LIN {X 0.186,Y -529.516,Z 604.576,A 0.000,B 0.000,C 90.000,E1 319.622} C_DIS
LIN {X -0.060,Y -530.503,Z 604.575,A 0.000,B 0.000,C 90.000,E1 319.504} C_DIS
LIN {X -0.169,Y -534.567,Z 604.573,A 0.000,B 0.000,C 90.000,E1 319.094} C_DIS
LIN {X -0.213,Y -539.708,Z 604.570,A 0.000,B 0.000,C 90.000,E1 318.609} C_DIS
LIN {X -0.061,Y -546.489,Z 604.567,A 0.000,B 0.000,C 90.000,E1 318.038} C_DIS
LIN {X 0.132,Y -560.853,Z 604.561,A 0.000,B 0.000,C 90.000,E1 316.905} C_DIS
LIN {X -0.105,Y -584.166,Z 604.551,A 0.000,B 0.000,C 90.000,E1 315.162} C_DIS
LIN {X -0.348,Y -592.593,Z 604.547,A 0.000,B 0.000,C 90.000,E1 314.514} C_DIS
LIN {X -0.144,Y -602.118,Z 604.543,A 0.000,B 0.000,C 90.000,E1 313.704} C_DIS
LIN {X -0.004,Y -608.600,Z 604.539,A 0.000,B 0.000,C 90.000,E1 313.095} C_DIS
LIN {X -0.128,Y -613.559,Z 604.537,A 0.000,B 0.000,C 90.000,E1 312.609} C_DIS
LIN {X 0.003,Y -618.325,Z 604.534,A 0.000,B 0.000,C 90.000,E1 312.081} C_DIS
LIN {X 0.217,Y -621.819,Z 604.532,A 0.000,B 0.000,C 90.000,E1 311.676} C_DIS
LIN {X -0.346,Y -626.177,Z 604.529,A 0.000,B 0.000,C 90.000,E1 311.229} C_DIS
LIN {X -0.271,Y -632.516,Z 604.525,A 0.000,B 0.000,C 90.000,E1 310.458} C_DIS
LIN {X 0.355,Y -638.703,Z 604.520,A 0.000,B 0.000,C 90.000,E1 309.644} C_DIS
LIN {X 0.149,Y -644.534,Z 604.516,A 0.000,B 0.000,C 90.000,E1 308.910} C_DIS
LIN {X -0.016,Y -649.070,Z 604.513,A 0.000,B 0.000,C 90.000,E1 308.302} C_DIS
LIN {X -0.079,Y -651.679,Z 604.511,A 0.000,B 0.000,C 90.000,E1 307.935} C_DIS
LIN {X -0.074,Y -655.621,Z 604.507,A 0.000,B 0.000,C 90.000,E1 307.317} C_DIS
LIN {X 0.328,Y -658.551,Z 604.505,A 0.000,B 0.000,C 90.000,E1 306.790} C_DIS
LIN {X -0.133,Y -661.855,Z 604.501,A 0.000,B 0.000,C 90.000,E1 306.217} C_DIS
LIN {X -0.035,Y -664.838,Z 604.498,A 0.000,B 0.000,C 90.000,E1 305.598} C_DIS
LIN {X -0.015,Y -668.105,Z 604.494,A 0.000,B 0.000,C 90.000,E1 304.865} C_DIS
LIN {X 0.202,Y -671.110,Z 604.490,A 0.000,B 0.000,C 90.000,E1 304.119} C_DIS
LIN {X 0.050,Y -674.814,Z 604.484,A 0.000,B 0.000,C 90.000,E1 303.166} C_DIS
LIN {X 0.125,Y -679.103,Z 604.478,A 0.000,B 0.000,C 90.000,E1 301.957} C_DIS
LIN {X -0.111,Y -684.040,Z 604.470,A 0.000,B 0.000,C 90.000,E1 300.541} C_DIS
LIN {X 0.330,Y -688.804,Z 604.462,A 0.000,B 0.000,C 90.000,E1 299.077} C_DIS
LIN {X -0.192,Y -691.108,Z 604.458,A 0.000,B 0.000,C 90.000,E1 298.409} C_DIS
LIN {X 0.081,Y -694.571,Z 604.451,A 0.000,B 0.000,C 90.000,E1 297.206} C_DIS
LIN {X -0.035,Y -695.805,Z 604.449,A 0.000,B 0.000,C 90.000,E1 296.744} C_DIS
LIN {X 0.219,Y -696.302,Z 604.447,A 0.000,B 0.000,C 90.000,E1 296.488} C_DIS
LIN {X 0.109,Y -696.935,Z 604.445,A 0.000,B 0.000,C 90.000,E1 296.027} C_DIS
LIN {X 0.064,Y -696.971,Z 604.443,A 0.000,B 0.000,C 90.000,E1 295.796} C_DIS
LIN {X -0.045,Y -696.271,Z 604.441,A 0.000,B 0.000,C 90.000,E1 295.335} C_DIS
LIN {X 0.212,Y -695.573,Z 604.439,A 0.000,B 0.000,C 90.000,E1 295.079} C_DIS
LIN {X -0.329,Y -693.248,Z 604.438,A 0.000,B 0.000,C 90.000,E1 294.771} C_DIS
LIN {X -0.202,Y -692.610,Z 604.437,A 0.000,B 0.000,C 90.000,E1 294.643} C_DIS
LIN {X -0.081,Y -691.776,Z 604.436,A 0.000,B 0.000,C 90.000,E1 294.515} C_DIS
LIN {X 0.042,Y -690.513,Z 604.436,A 0.000,B 0.000,C 90.000,E1 294.387} C_DIS
LIN {X 0.205,Y -688.584,Z 604.435,A 0.000,B 0.000,C 90.000,E1 294.259} C_DIS
LIN {X -0.053,Y -683.886,Z 604.434,A 0.000,B 0.000,C 90.000,E1 294.027} C_DIS
LIN {X -0.165,Y -682.015,Z 604.433,A 0.000,B 0.000,C 90.000,E1 293.951} C_DIS
LIN {X -0.285,Y -677.558,Z 604.432,A 0.000,B 0.000,C 90.000,E1 293.823} C_DIS
LIN {X -0.294,Y -675.531,Z 604.432,A 0.000,B 0.000,C 90.000,E1 293.770} C_DIS
LIN {X -0.285,Y -668.871,Z 604.431,A 0.000,B 0.000,C 90.000,E1 293.643} C_DIS
LIN {X 0.110,Y -658.714,Z 604.430,A 0.000,B 0.000,C 90.000,E1 293.462} C_DIS
LIN {X -0.016,Y -648.477,Z 604.430,A 0.000,B 0.000,C 90.000,E1 293.334} C_DIS
LIN {X 0.187,Y -635.246,Z 604.428,A 0.000,B 0.000,C 90.000,E1 293.078} C_DIS
LIN {X 0.120,Y -629.181,Z 604.428,A 0.000,B 0.000,C 90.000,E1 292.950} C_DIS
LIN {X 0.085,Y -619.069,Z 604.426,A 0.000,B 0.000,C 90.000,E1 292.695} C_DIS
LIN {X 0.147,Y -598.743,Z 604.423,A 0.000,B 0.000,C 90.000,E1 292.078} C_DIS
LIN {X 0.201,Y -579.627,Z 604.419,A 0.000,B 0.000,C 90.000,E1 291.461} C_DIS
LIN {X -0.020,Y -570.715,Z 604.418,A 0.000,B 0.000,C 90.000,E1 291.227} C_DIS
LIN {X -0.270,Y -566.103,Z 604.417,A 0.000,B 0.000,C 90.000,E1 291.099} C_DIS
LIN {X 0.225,Y -563.210,Z 604.416,A 0.000,B 0.000,C 90.000,E1 290.918} C_DIS
LIN {X -0.054,Y -560.151,Z 604.416,A 0.000,B 0.000,C 90.000,E1 290.791} C_DIS
LIN {X -0.106,Y -560.098,Z 604.415,A 0.000,B 0.000,C 90.000,E1 290.791} C_DIS
LIN {X 0.099,Y -558.817,Z 604.415,A 0.000,B 0.000,C 90.000,E1 290.610} C_DIS
LIN {X 0.055,Y -558.800,Z 604.415,A 0.000,B 0.000,C 90.000,E1 290.610} C_DIS
LIN {X -0.102,Y -558.249,Z 604.413,A 0.000,B 0.000,C 90.000,E1 290.355} C_DIS
LIN {X 0.244,Y -558.020,Z 604.408,A 0.000,B 0.000,C 90.000,E1 289.450} C_DIS
LIN {X 0.015,Y -558.055,Z 604.402,A 0.000,B 0.000,C 90.000,E1 288.362} C_DIS
LIN {X 0.192,Y -557.907,Z 604.397,A 0.000,B 0.000,C 90.000,E1 287.511} C_DIS
LIN {X 0.079,Y -557.543,Z 604.390,A 0.000,B 0.000,C 90.000,E1 286.134} C_DIS
LIN {X -0.194,Y -556.910,Z 604.382,A 0.000,B 0.000,C 90.000,E1 284.773} C_DIS
LIN {X 0.066,Y -556.250,Z 604.374,A 0.000,B 0.000,C 90.000,E1 283.355} C_DIS
LIN {X 0.190,Y -555.485,Z 604.367,A 0.000,B 0.000,C 90.000,E1 281.951} C_DIS
LIN {X 0.012,Y -554.480,Z 604.356,A 0.000,B 0.000,C 90.000,E1 280.018} C_DIS
LIN {X 0.159,Y -553.428,Z 604.345,A 0.000,B 0.000,C 90.000,E1 278.049} C_DIS
LIN {X -0.227,Y -552.417,Z 604.332,A 0.000,B 0.000,C 90.000,E1 275.853} C_DIS
LIN {X -0.261,Y -551.657,Z 604.322,A 0.000,B 0.000,C 90.000,E1 273.898} C_DIS
LIN {X 0.176,Y -551.113,Z 604.311,A 0.000,B 0.000,C 90.000,E1 271.892} C_DIS
LIN {X -0.004,Y -550.680,Z 604.301,A 0.000,B 0.000,C 90.000,E1 270.229} C_DIS
LIN {X 0.229,Y -550.313,Z 604.295,A 0.000,B 0.000,C 90.000,E1 269.083} C_DIS
LIN {X -0.026,Y -549.760,Z 604.287,A 0.000,B 0.000,C 90.000,E1 267.707} C_DIS
LIN {X -0.242,Y -549.027,Z 604.278,A 0.000,B 0.000,C 90.000,E1 266.045} C_DIS
LIN {X 0.056,Y -548.306,Z 604.270,A 0.000,B 0.000,C 90.000,E1 264.609} C_DIS
LIN {X -0.240,Y -547.656,Z 604.264,A 0.000,B 0.000,C 90.000,E1 263.514} C_DIS
LIN {X 0.066,Y -546.707,Z 604.258,A 0.000,B 0.000,C 90.000,E1 262.356} C_DIS
LIN {X -0.167,Y -545.476,Z 604.250,A 0.000,B 0.000,C 90.000,E1 260.971} C_DIS
LIN {X -0.170,Y -543.553,Z 604.239,A 0.000,B 0.000,C 90.000,E1 258.993} C_DIS
LIN {X -0.081,Y -541.959,Z 604.229,A 0.000,B 0.000,C 90.000,E1 257.285} C_DIS
LIN {X -0.217,Y -540.569,Z 604.221,A 0.000,B 0.000,C 90.000,E1 255.880} C_DIS
LIN {X -0.117,Y -539.138,Z 604.214,A 0.000,B 0.000,C 90.000,E1 254.448} C_DIS
LIN {X -0.035,Y -537.671,Z 604.206,A 0.000,B 0.000,C 90.000,E1 253.015} C_DIS
LIN {X 0.012,Y -536.182,Z 604.198,A 0.000,B 0.000,C 90.000,E1 251.583} C_DIS
LIN {X 0.163,Y -534.919,Z 604.191,A 0.000,B 0.000,C 90.000,E1 250.423} C_DIS
LIN {X 0.299,Y -533.212,Z 604.185,A 0.000,B 0.000,C 90.000,E1 249.263} C_DIS
LIN {X -0.089,Y -531.283,Z 604.179,A 0.000,B 0.000,C 90.000,E1 248.156} C_DIS
LIN {X 0.189,Y -529.215,Z 604.172,A 0.000,B 0.000,C 90.000,E1 246.975} C_DIS
LIN {X 0.127,Y -526.472,Z 604.164,A 0.000,B 0.000,C 90.000,E1 245.537} C_DIS
LIN {X 0.156,Y -524.679,Z 604.159,A 0.000,B 0.000,C 90.000,E1 244.665} C_DIS
LIN {X -0.246,Y -521.576,Z 604.151,A 0.000,B 0.000,C 90.000,E1 243.256} C_DIS
LIN {X -0.001,Y -518.258,Z 604.143,A 0.000,B 0.000,C 90.000,E1 241.769} C_DIS
LIN {X 0.066,Y -515.423,Z 604.137,A 0.000,B 0.000,C 90.000,E1 240.589} C_DIS
LIN {X -0.015,Y -510.401,Z 604.125,A 0.000,B 0.000,C 90.000,E1 238.535} C_DIS
LIN {X -0.140,Y -508.226,Z 604.120,A 0.000,B 0.000,C 90.000,E1 237.661} C_DIS
LIN {X -0.014,Y -505.922,Z 604.115,A 0.000,B 0.000,C 90.000,E1 236.755} C_DIS
LIN {X 0.113,Y -502.599,Z 604.109,A 0.000,B 0.000,C 90.000,E1 235.548} C_DIS
LIN {X 0.236,Y -495.945,Z 604.095,A 0.000,B 0.000,C 90.000,E1 233.130} C_DIS
LIN {X 0.228,Y -492.067,Z 604.087,A 0.000,B 0.000,C 90.000,E1 231.618} C_DIS
LIN {X -0.078,Y -488.885,Z 604.080,A 0.000,B 0.000,C 90.000,E1 230.436} C_DIS
LIN {X -0.114,Y -485.802,Z 604.073,A 0.000,B 0.000,C 90.000,E1 229.218} C_DIS
LIN {X 0.004,Y -479.575,Z 604.060,A 0.000,B 0.000,C 90.000,E1 226.743} C_DIS
LIN {X 0.038,Y -475.057,Z 604.049,A 0.000,B 0.000,C 90.000,E1 224.879} C_DIS
LIN {X -0.121,Y -471.425,Z 604.041,A 0.000,B 0.000,C 90.000,E1 223.338} C_DIS
LIN {X -0.096,Y -468.638,Z 604.034,A 0.000,B 0.000,C 90.000,E1 222.081} C_DIS
LIN {X 0.257,Y -462.337,Z 604.018,A 0.000,B 0.000,C 90.000,E1 219.197} C_DIS
LIN {X 0.025,Y -458.399,Z 604.007,A 0.000,B 0.000,C 90.000,E1 217.317} C_DIS
LIN {X 0.073,Y -454.602,Z 603.997,A 0.000,B 0.000,C 90.000,E1 215.391} C_DIS
LIN {X 0.019,Y -449.126,Z 603.981,A 0.000,B 0.000,C 90.000,E1 212.498} C_DIS
LIN {X 0.093,Y -445.604,Z 603.970,A 0.000,B 0.000,C 90.000,E1 210.541} C_DIS
LIN {X -0.149,Y -442.083,Z 603.959,A 0.000,B 0.000,C 90.000,E1 208.615} C_DIS
LIN {X 0.052,Y -439.190,Z 603.950,A 0.000,B 0.000,C 90.000,E1 206.950} C_DIS
LIN {X -0.026,Y -436.899,Z 603.943,A 0.000,B 0.000,C 90.000,E1 205.643} C_DIS
LIN {X -0.122,Y -434.073,Z 603.933,A 0.000,B 0.000,C 90.000,E1 204.003} C_DIS
LIN {X -0.014,Y -430.197,Z 603.920,A 0.000,B 0.000,C 90.000,E1 201.663} C_DIS
LIN {X -0.011,Y -426.364,Z 603.907,A 0.000,B 0.000,C 90.000,E1 199.322} C_DIS
LIN {X 0.053,Y -422.331,Z 603.892,A 0.000,B 0.000,C 90.000,E1 196.622} C_DIS
LIN {X 0.058,Y -419.574,Z 603.881,A 0.000,B 0.000,C 90.000,E1 194.592} C_DIS
LIN {X 0.134,Y -417.051,Z 603.872,A 0.000,B 0.000,C 90.000,E1 192.883} C_DIS
LIN {X 0.023,Y -414.987,Z 603.864,A 0.000,B 0.000,C 90.000,E1 191.535} C_DIS
LIN {X -0.007,Y -410.857,Z 603.847,A 0.000,B 0.000,C 90.000,E1 188.454} C_DIS
LIN {X 0.055,Y -409.129,Z 603.839,A 0.000,B 0.000,C 90.000,E1 187.068} C_DIS
LIN {X 0.080,Y -406.021,Z 603.826,A 0.000,B 0.000,C 90.000,E1 184.645} C_DIS
LIN {X 0.154,Y -401.641,Z 603.803,A 0.000,B 0.000,C 90.000,E1 180.458} C_DIS
LIN {X 0.087,Y -398.904,Z 603.781,A 0.000,B 0.000,C 90.000,E1 176.617} C_DIS
LIN {X 0.041,Y -397.580,Z 603.762,A 0.000,B 0.000,C 90.000,E1 173.109} C_DIS
LIN {X -0.213,Y -397.041,Z 603.746,A 0.000,B 0.000,C 90.000,E1 170.330} C_DIS
LIN {X 0.091,Y -397.075,Z 603.729,A 0.000,B 0.000,C 90.000,E1 167.117} C_DIS
LIN {X -0.026,Y -397.756,Z 603.709,A 0.000,B 0.000,C 90.000,E1 163.614} C_DIS
LIN {X 0.002,Y -398.448,Z 603.695,A 0.000,B 0.000,C 90.000,E1 161.148} C_DIS
LIN {X 0.088,Y -399.125,Z 603.684,A 0.000,B 0.000,C 90.000,E1 159.028} C_DIS
LIN {X -0.195,Y -400.052,Z 603.670,A 0.000,B 0.000,C 90.000,E1 156.613} C_DIS
LIN {X 0.051,Y -400.640,Z 603.662,A 0.000,B 0.000,C 90.000,E1 155.177} C_DIS
LIN {X -0.058,Y -401.693,Z 603.649,A 0.000,B 0.000,C 90.000,E1 152.743} C_DIS
LIN {X -0.091,Y -402.339,Z 603.639,A 0.000,B 0.000,C 90.000,E1 151.001} C_DIS
LIN {X -0.067,Y -402.941,Z 603.629,A 0.000,B 0.000,C 90.000,E1 149.253} C_DIS
LIN {X -0.019,Y -403.487,Z 603.620,A 0.000,B 0.000,C 90.000,E1 147.502} C_DIS
LIN {X 0.152,Y -404.062,Z 603.608,A 0.000,B 0.000,C 90.000,E1 145.388} C_DIS
LIN {X -0.235,Y -404.521,Z 603.598,A 0.000,B 0.000,C 90.000,E1 143.703} C_DIS
LIN {X -0.241,Y -405.187,Z 603.587,A 0.000,B 0.000,C 90.000,E1 141.618} C_DIS
LIN {X -0.005,Y -405.631,Z 603.579,A 0.000,B 0.000,C 90.000,E1 140.194} C_DIS
LIN {X 0.077,Y -406.094,Z 603.569,A 0.000,B 0.000,C 90.000,E1 138.447} C_DIS
LIN {X -0.003,Y -406.469,Z 603.558,A 0.000,B 0.000,C 90.000,E1 136.377} C_DIS
LIN {X -0.229,Y -406.760,Z 603.548,A 0.000,B 0.000,C 90.000,E1 134.676} C_DIS
LIN {X 0.260,Y -407.085,Z 603.536,A 0.000,B 0.000,C 90.000,E1 132.528} C_DIS
LIN {X 0.202,Y -407.379,Z 603.525,A 0.000,B 0.000,C 90.000,E1 130.458} C_DIS
LIN {X 0.005,Y -407.740,Z 603.515,A 0.000,B 0.000,C 90.000,E1 128.669} C_DIS
LIN {X -0.085,Y -415.448,Z 603.500,A 0.000,B 0.000,C 90.000,E1 126.011} C_DIS
LIN {X -0.089,Y -423.340,Z 603.482,A 0.000,B 0.000,C 90.000,E1 122.832} C_DIS
LIN {X -0.129,Y -423.366,Z 603.482,A 0.000,B 0.000,C 90.000,E1 122.832} C_DIS
LIN {X 0.085,Y -428.902,Z 603.481,A 0.000,B 0.000,C 90.000,E1 122.498} C_DIS
LIN {X -0.125,Y -446.238,Z 603.476,A 0.000,B 0.000,C 90.000,E1 121.671} C_DIS
LIN {X -0.196,Y -454.719,Z 603.474,A 0.000,B 0.000,C 90.000,E1 121.258} C_DIS
LIN {X 0.127,Y -461.547,Z 603.472,A 0.000,B 0.000,C 90.000,E1 120.875} C_DIS
LIN {X 0.022,Y -473.001,Z 603.468,A 0.000,B 0.000,C 90.000,E1 120.256} C_DIS
LIN {X -0.058,Y -481.216,Z 603.466,A 0.000,B 0.000,C 90.000,E1 119.795} C_DIS
LIN {X -0.136,Y -487.657,Z 603.463,A 0.000,B 0.000,C 90.000,E1 119.411} C_DIS
LIN {X -0.317,Y -497.266,Z 603.460,A 0.000,B 0.000,C 90.000,E1 118.821} C_DIS
LIN {X 0.190,Y -505.096,Z 603.457,A 0.000,B 0.000,C 90.000,E1 118.231} C_DIS
LIN {X -0.161,Y -512.793,Z 603.454,A 0.000,B 0.000,C 90.000,E1 117.719} C_DIS
LIN {X -0.067,Y -518.829,Z 603.451,A 0.000,B 0.000,C 90.000,E1 117.257} C_DIS
LIN {X 0.054,Y -527.774,Z 603.448,A 0.000,B 0.000,C 90.000,E1 116.539} C_DIS
LIN {X 0.156,Y -533.532,Z 603.445,A 0.000,B 0.000,C 90.000,E1 116.052} C_DIS
LIN {X 0.031,Y -539.012,Z 603.442,A 0.000,B 0.000,C 90.000,E1 115.591} C_DIS
LIN {X -0.185,Y -544.084,Z 603.440,A 0.000,B 0.000,C 90.000,E1 115.155} C_DIS
LIN {X -0.136,Y -548.015,Z 603.438,A 0.000,B 0.000,C 90.000,E1 114.771} C_DIS
LIN {X -0.187,Y -550.349,Z 603.436,A 0.000,B 0.000,C 90.000,E1 114.515} C_DIS
LIN {X 0.193,Y -551.795,Z 603.435,A 0.000,B 0.000,C 90.000,E1 114.335} C_DIS
LIN {X 0.000,Y -553.592,Z 603.434,A 0.000,B 0.000,C 90.000,E1 114.155} C_DIS
LIN {X -0.087,Y -557.876,Z 603.431,A 0.000,B 0.000,C 90.000,E1 113.643} C_DIS
LIN {X 0.206,Y -559.765,Z 603.430,A 0.000,B 0.000,C 90.000,E1 113.334} C_DIS
LIN {X 0.333,Y -562.532,Z 603.428,A 0.000,B 0.000,C 90.000,E1 112.950} C_DIS
LIN {X 0.137,Y -566.836,Z 603.424,A 0.000,B 0.000,C 90.000,E1 112.280} C_DIS
LIN {X 0.105,Y -571.305,Z 603.419,A 0.000,B 0.000,C 90.000,E1 111.461} C_DIS
LIN {X -0.098,Y -575.474,Z 603.415,A 0.000,B 0.000,C 90.000,E1 110.663} C_DIS
LIN {X -0.095,Y -578.012,Z 603.412,A 0.000,B 0.000,C 90.000,E1 110.120} C_DIS
LIN {X -0.237,Y -581.484,Z 603.407,A 0.000,B 0.000,C 90.000,E1 109.322} C_DIS
LIN {X 0.017,Y -584.659,Z 603.403,A 0.000,B 0.000,C 90.000,E1 108.489} C_DIS
LIN {X 0.088,Y -586.670,Z 603.400,A 0.000,B 0.000,C 90.000,E1 107.946} C_DIS
LIN {X 0.023,Y -589.389,Z 603.395,A 0.000,B 0.000,C 90.000,E1 107.149} C_DIS
LIN {X 0.061,Y -592.616,Z 603.389,A 0.000,B 0.000,C 90.000,E1 106.079} C_DIS
LIN {X -0.150,Y -596.388,Z 603.382,A 0.000,B 0.000,C 90.000,E1 104.773} C_DIS
LIN {X -0.003,Y -601.209,Z 603.373,A 0.000,B 0.000,C 90.000,E1 103.175} C_DIS
LIN {X 0.101,Y -606.068,Z 603.365,A 0.000,B 0.000,C 90.000,E1 101.591} C_DIS
LIN {X 0.110,Y -609.345,Z 603.359,A 0.000,B 0.000,C 90.000,E1 100.546} C_DIS
LIN {X 0.171,Y -612.516,Z 603.353,A 0.000,B 0.000,C 90.000,E1 99.500} C_DIS
LIN {X 0.026,Y -616.220,Z 603.346,A 0.000,B 0.000,C 90.000,E1 98.219} C_DIS
LIN {X 0.139,Y -620.381,Z 603.337,A 0.000,B 0.000,C 90.000,E1 96.663} C_DIS
LIN {X -0.045,Y -622.372,Z 603.333,A 0.000,B 0.000,C 90.000,E1 95.910} C_DIS
LIN {X -0.198,Y -625.198,Z 603.326,A 0.000,B 0.000,C 90.000,E1 94.645} C_DIS
LIN {X -0.158,Y -626.245,Z 603.323,A 0.000,B 0.000,C 90.000,E1 94.131} C_DIS
LIN {X -0.249,Y -628.469,Z 603.316,A 0.000,B 0.000,C 90.000,E1 92.865} C_DIS
LIN {X -0.093,Y -630.019,Z 603.310,A 0.000,B 0.000,C 90.000,E1 91.835} C_DIS
LIN {X -0.258,Y -631.003,Z 603.306,A 0.000,B 0.000,C 90.000,E1 91.088} C_DIS
LIN {X -0.061,Y -632.004,Z 603.300,A 0.000,B 0.000,C 90.000,E1 90.057} C_DIS
LIN {X 0.148,Y -632.628,Z 603.295,A 0.000,B 0.000,C 90.000,E1 89.026} C_DIS
LIN {X -0.252,Y -632.868,Z 603.289,A 0.000,B 0.000,C 90.000,E1 88.051} C_DIS
LIN {X -0.040,Y -632.700,Z 603.283,A 0.000,B 0.000,C 90.000,E1 87.020} C_DIS
LIN {X 0.095,Y -632.540,Z 603.281,A 0.000,B 0.000,C 90.000,E1 86.502} C_DIS
LIN {X -0.303,Y -631.955,Z 603.275,A 0.000,B 0.000,C 90.000,E1 85.527} C_DIS
LIN {X -0.026,Y -631.135,Z 603.269,A 0.000,B 0.000,C 90.000,E1 84.489} C_DIS
LIN {X 0.173,Y -630.107,Z 603.264,A 0.000,B 0.000,C 90.000,E1 83.457} C_DIS
LIN {X 0.086,Y -629.130,Z 603.260,A 0.000,B 0.000,C 90.000,E1 82.704} C_DIS
LIN {X -0.306,Y -627.479,Z 603.254,A 0.000,B 0.000,C 90.000,E1 81.724} C_DIS
LIN {X 0.202,Y -626.153,Z 603.250,A 0.000,B 0.000,C 90.000,E1 80.914} C_DIS
LIN {X 0.261,Y -623.569,Z 603.243,A 0.000,B 0.000,C 90.000,E1 79.634} C_DIS
LIN {X -0.210,Y -620.708,Z 603.235,A 0.000,B 0.000,C 90.000,E1 78.398} C_DIS
LIN {X -0.014,Y -618.279,Z 603.230,A 0.000,B 0.000,C 90.000,E1 77.353} C_DIS
LIN {X 0.035,Y -614.902,Z 603.223,A 0.000,B 0.000,C 90.000,E1 76.061} C_DIS
LIN {X -0.172,Y -611.974,Z 603.217,A 0.000,B 0.000,C 90.000,E1 75.046} C_DIS
LIN {X -0.157,Y -609.699,Z 603.213,A 0.000,B 0.000,C 90.000,E1 74.267} C_DIS
LIN {X -0.333,Y -607.231,Z 603.208,A 0.000,B 0.000,C 90.000,E1 73.504} C_DIS
LIN {X 0.211,Y -604.497,Z 603.204,A 0.000,B 0.000,C 90.000,E1 72.670} C_DIS
LIN {X 0.144,Y -601.468,Z 603.200,A 0.000,B 0.000,C 90.000,E1 71.891} C_DIS
LIN {X 0.237,Y -598.125,Z 603.195,A 0.000,B 0.000,C 90.000,E1 71.094} C_DIS
LIN {X 0.355,Y -595.172,Z 603.191,A 0.000,B 0.000,C 90.000,E1 70.423} C_DIS
LIN {X 0.067,Y -590.089,Z 603.186,A 0.000,B 0.000,C 90.000,E1 69.390} C_DIS
LIN {X 0.170,Y -587.424,Z 603.183,A 0.000,B 0.000,C 90.000,E1 68.847} C_DIS
LIN {X -0.143,Y -583.796,Z 603.179,A 0.000,B 0.000,C 90.000,E1 68.209} C_DIS
LIN {X -0.105,Y -579.955,Z 603.175,A 0.000,B 0.000,C 90.000,E1 67.539} C_DIS
LIN {X -0.107,Y -575.682,Z 603.172,A 0.000,B 0.000,C 90.000,E1 66.869} C_DIS
LIN {X 0.023,Y -570.882,Z 603.168,A 0.000,B 0.000,C 90.000,E1 66.177} C_DIS
LIN {X 0.201,Y -566.749,Z 603.165,A 0.000,B 0.000,C 90.000,E1 65.613} C_DIS
LIN {X -0.163,Y -562.256,Z 603.162,A 0.000,B 0.000,C 90.000,E1 65.101} C_DIS
LIN {X -0.023,Y -557.404,Z 603.159,A 0.000,B 0.000,C 90.000,E1 64.537} C_DIS
LIN {X -0.232,Y -552.136,Z 603.156,A 0.000,B 0.000,C 90.000,E1 64.024} C_DIS
LIN {X 0.125,Y -546.904,Z 603.153,A 0.000,B 0.000,C 90.000,E1 63.512} C_DIS
LIN {X 0.040,Y -541.354,Z 603.151,A 0.000,B 0.000,C 90.000,E1 63.076} C_DIS
LIN {X 0.072,Y -535.391,Z 603.148,A 0.000,B 0.000,C 90.000,E1 62.666} C_DIS
LIN {X 0.108,Y -530.416,Z 603.147,A 0.000,B 0.000,C 90.000,E1 62.359} C_DIS
LIN {X -0.019,Y -520.380,Z 603.143,A 0.000,B 0.000,C 90.000,E1 61.820} C_DIS
LIN {X 0.156,Y -512.066,Z 603.141,A 0.000,B 0.000,C 90.000,E1 61.385} C_DIS
LIN {X -0.034,Y -500.016,Z 603.138,A 0.000,B 0.000,C 90.000,E1 60.845} C_DIS
LIN {X 0.255,Y -477.828,Z 603.132,A 0.000,B 0.000,C 90.000,E1 59.793} C_DIS
LIN {X 0.036,Y -472.634,Z 603.131,A 0.000,B 0.000,C 90.000,E1 59.587} C_DIS
LIN {X -0.170,Y -447.331,Z 603.124,A 0.000,B 0.000,C 90.000,E1 58.329} C_DIS
LIN {X -0.212,Y -447.300,Z 603.124,A 0.000,B 0.000,C 90.000,E1 58.329} C_DIS
LIN {X -0.059,Y -444.169,Z 603.115,A 0.000,B 0.000,C 90.000,E1 56.628} C_DIS
LIN {X 0.054,Y -442.600,Z 603.111,A 0.000,B 0.000,C 90.000,E1 55.960} C_DIS
LIN {X -0.084,Y -433.734,Z 603.089,A 0.000,B 0.000,C 90.000,E1 52.029} C_DIS
LIN {X 0.090,Y -431.207,Z 603.082,A 0.000,B 0.000,C 90.000,E1 50.678} C_DIS
LIN {X -0.029,Y -431.072,Z 603.081,A 0.000,B 0.000,C 90.000,E1 50.642} C_DIS
LIN {X -0.067,Y -431.069,Z 603.081,A 0.000,B 0.000,C 90.000,E1 50.642} C_DIS
LIN {X -0.166,Y -431.992,Z 603.074,A 0.000,B 0.000,C 90.000,E1 49.380} C_DIS
LIN {X -0.150,Y -433.088,Z 603.065,A 0.000,B 0.000,C 90.000,E1 47.715} C_DIS
LIN {X -0.024,Y -433.733,Z 603.060,A 0.000,B 0.000,C 90.000,E1 46.701} C_DIS
LIN {X 0.190,Y -435.220,Z 603.047,A 0.000,B 0.000,C 90.000,E1 44.352} C_DIS
LIN {X -0.024,Y -436.123,Z 603.039,A 0.000,B 0.000,C 90.000,E1 43.056} C_DIS
LIN {X -0.205,Y -436.865,Z 603.032,A 0.000,B 0.000,C 90.000,E1 41.757} C_DIS
LIN {X -0.092,Y -437.734,Z 603.023,A 0.000,B 0.000,C 90.000,E1 40.092} C_DIS
LIN {X 0.042,Y -438.590,Z 603.012,A 0.000,B 0.000,C 90.000,E1 38.096} C_DIS
LIN {X -0.042,Y -438.993,Z 603.004,A 0.000,B 0.000,C 90.000,E1 36.790} C_DIS
LIN {X -0.025,Y -439.354,Z 602.997,A 0.000,B 0.000,C 90.000,E1 35.471} C_DIS
LIN {X 0.253,Y -439.632,Z 602.990,A 0.000,B 0.000,C 90.000,E1 34.119} C_DIS
LIN {X 0.039,Y -439.838,Z 602.982,A 0.000,B 0.000,C 90.000,E1 32.832} C_DIS
LIN {X -0.124,Y -440.034,Z 602.973,A 0.000,B 0.000,C 90.000,E1 31.209} C_DIS
LIN {X 0.089,Y -440.296,Z 602.964,A 0.000,B 0.000,C 90.000,E1 29.539} C_DIS
LIN {X 0.044,Y -440.508,Z 602.957,A 0.000,B 0.000,C 90.000,E1 28.231} C_DIS
LIN {X -0.003,Y -440.751,Z 602.950,A 0.000,B 0.000,C 90.000,E1 26.924} C_DIS
LIN {X 0.023,Y -441.108,Z 602.939,A 0.000,B 0.000,C 90.000,E1 24.951} C_DIS
LIN {X -0.005,Y -441.428,Z 602.931,A 0.000,B 0.000,C 90.000,E1 23.643} C_DIS
LIN {X -0.171,Y -441.892,Z 602.922,A 0.000,B 0.000,C 90.000,E1 22.025} C_DIS
LIN {X -0.226,Y -442.467,Z 602.911,A 0.000,B 0.000,C 90.000,E1 20.066} C_DIS
LIN {X -0.140,Y -443.208,Z 602.899,A 0.000,B 0.000,C 90.000,E1 17.764} C_DIS
LIN {X -0.180,Y -444.134,Z 602.886,A 0.000,B 0.000,C 90.000,E1 15.481} C_DIS
LIN {X 0.156,Y -445.442,Z 602.871,A 0.000,B 0.000,C 90.000,E1 12.827} C_DIS
LIN {X -0.165,Y -447.553,Z 602.853,A 0.000,B 0.000,C 90.000,E1 9.613} C_DIS
LIN {X 0.189,Y -449.250,Z 602.841,A 0.000,B 0.000,C 90.000,E1 7.296} C_DIS
LIN {X 0.037,Y -451.202,Z 602.828,A 0.000,B 0.000,C 90.000,E1 5.049} C_DIS
LIN {X 0.184,Y -453.147,Z 602.817,A 0.000,B 0.000,C 90.000,E1 3.094} C_DIS
LIN {X 0.047,Y -455.600,Z 602.805,A 0.000,B 0.000,C 90.000,E1 0.859} C_DIS
LIN {X 0.012,Y -458.664,Z 602.792,A 0.000,B 0.000,C 90.000,E1 358.511} C_DIS
LIN {X -0.236,Y -463.332,Z 602.774,A 0.000,B 0.000,C 90.000,E1 355.355} C_DIS
LIN {X 0.001,Y -466.846,Z 602.762,A 0.000,B 0.000,C 90.000,E1 353.109} C_DIS
LIN {X 0.087,Y -468.874,Z 602.755,A 0.000,B 0.000,C 90.000,E1 351.837} C_DIS
LIN {X -0.155,Y -471.796,Z 602.744,A 0.000,B 0.000,C 90.000,E1 349.982} C_DIS
LIN {X -0.182,Y -476.487,Z 602.729,A 0.000,B 0.000,C 90.000,E1 347.173} C_DIS
LIN {X 0.039,Y -479.782,Z 602.718,A 0.000,B 0.000,C 90.000,E1 345.283} C_DIS
LIN {X 0.002,Y -483.212,Z 602.708,A 0.000,B 0.000,C 90.000,E1 343.433} C_DIS
LIN {X 0.037,Y -486.676,Z 602.698,A 0.000,B 0.000,C 90.000,E1 341.583} C_DIS
LIN {X -0.035,Y -489.672,Z 602.689,A 0.000,B 0.000,C 90.000,E1 340.061} C_DIS
LIN {X -0.054,Y -492.540,Z 602.681,A 0.000,B 0.000,C 90.000,E1 338.539} C_DIS
LIN {X 0.109,Y -494.749,Z 602.674,A 0.000,B 0.000,C 90.000,E1 337.305} C_DIS
LIN {X 0.155,Y -497.768,Z 602.664,A 0.000,B 0.000,C 90.000,E1 335.485} C_DIS
LIN {X 0.036,Y -500.588,Z 602.654,A 0.000,B 0.000,C 90.000,E1 333.691} C_DIS
LIN {X 0.065,Y -502.387,Z 602.647,A 0.000,B 0.000,C 90.000,E1 332.487} C_DIS
LIN {X -0.163,Y -505.067,Z 602.637,A 0.000,B 0.000,C 90.000,E1 330.717} C_DIS
LIN {X -0.076,Y -507.735,Z 602.627,A 0.000,B 0.000,C 90.000,E1 328.918} C_DIS
LIN {X -0.118,Y -511.655,Z 602.614,A 0.000,B 0.000,C 90.000,E1 326.548} C_DIS
LIN {X -0.124,Y -515.571,Z 602.603,A 0.000,B 0.000,C 90.000,E1 324.482} C_DIS
LIN {X -0.104,Y -519.152,Z 602.593,A 0.000,B 0.000,C 90.000,E1 322.718} C_DIS
LIN {X -0.058,Y -522.242,Z 602.585,A 0.000,B 0.000,C 90.000,E1 321.251} C_DIS
LIN {X 0.034,Y -523.415,Z 602.582,A 0.000,B 0.000,C 90.000,E1 320.803} C_DIS
LIN {X -0.007,Y -525.171,Z 602.580,A 0.000,B 0.000,C 90.000,E1 320.312} C_DIS
LIN {X 0.139,Y -525.650,Z 602.579,A 0.000,B 0.000,C 90.000,E1 320.150} C_DIS
LIN {X 0.227,Y -527.273,Z 602.577,A 0.000,B 0.000,C 90.000,E1 319.828} C_DIS
LIN {X 0.038,Y -527.840,Z 602.576,A 0.000,B 0.000,C 90.000,E1 319.703} C_DIS
LIN {X 0.192,Y -528.600,Z 602.575,A 0.000,B 0.000,C 90.000,E1 319.542} C_DIS
LIN {X -0.239,Y -530.451,Z 602.574,A 0.000,B 0.000,C 90.000,E1 319.299} C_DIS
LIN {X -0.080,Y -531.166,Z 602.573,A 0.000,B 0.000,C 90.000,E1 319.138} C_DIS
LIN {X 0.002,Y -531.663,Z 602.573,A 0.000,B 0.000,C 90.000,E1 319.057} C_DIS
LIN {X 0.042,Y -537.684,Z 602.569,A 0.000,B 0.000,C 90.000,E1 318.447} C_DIS
LIN {X 0.118,Y -543.184,Z 602.567,A 0.000,B 0.000,C 90.000,E1 317.957} C_DIS
LIN {X -0.165,Y -559.196,Z 602.560,A 0.000,B 0.000,C 90.000,E1 316.743} C_DIS
LIN {X 0.271,Y -582.714,Z 602.550,A 0.000,B 0.000,C 90.000,E1 314.919} C_DIS
LIN {X -0.183,Y -592.665,Z 602.545,A 0.000,B 0.000,C 90.000,E1 314.190} C_DIS
LIN {X -0.062,Y -602.383,Z 602.541,A 0.000,B 0.000,C 90.000,E1 313.380} C_DIS
LIN {X 0.092,Y -607.542,Z 602.538,A 0.000,B 0.000,C 90.000,E1 312.894} C_DIS
LIN {X 0.045,Y -612.513,Z 602.536,A 0.000,B 0.000,C 90.000,E1 312.405} C_DIS
LIN {X 0.079,Y -619.818,Z 602.531,A 0.000,B 0.000,C 90.000,E1 311.634} C_DIS
LIN {X -0.229,Y -624.385,Z 602.529,A 0.000,B 0.000,C 90.000,E1 311.148} C_DIS
LIN {X 0.339,Y -629.720,Z 602.525,A 0.000,B 0.000,C 90.000,E1 310.458} C_DIS
LIN {X -0.282,Y -636.948,Z 602.520,A 0.000,B 0.000,C 90.000,E1 309.644} C_DIS
LIN {X -0.008,Y -641.895,Z 602.517,A 0.000,B 0.000,C 90.000,E1 308.991} C_DIS
LIN {X -0.184,Y -647.529,Z 602.513,A 0.000,B 0.000,C 90.000,E1 308.257} C_DIS
LIN {X 0.165,Y -651.004,Z 602.510,A 0.000,B 0.000,C 90.000,E1 307.729} C_DIS
LIN {X -0.354,Y -655.026,Z 602.506,A 0.000,B 0.000,C 90.000,E1 307.156} C_DIS
LIN {X -0.353,Y -657.929,Z 602.504,A 0.000,B 0.000,C 90.000,E1 306.664} C_DIS
LIN {X 0.058,Y -660.645,Z 602.501,A 0.000,B 0.000,C 90.000,E1 306.137} C_DIS
LIN {X 0.097,Y -663.148,Z 602.498,A 0.000,B 0.000,C 90.000,E1 305.644} C_DIS
LIN {X 0.263,Y -666.529,Z 602.494,A 0.000,B 0.000,C 90.000,E1 304.898} C_DIS
LIN {X -0.082,Y -669.659,Z 602.490,A 0.000,B 0.000,C 90.000,E1 304.199} C_DIS
LIN {X 0.117,Y -673.466,Z 602.485,A 0.000,B 0.000,C 90.000,E1 303.214} C_DIS
LIN {X -0.236,Y -678.690,Z 602.477,A 0.000,B 0.000,C 90.000,E1 301.799} C_DIS
LIN {X 0.097,Y -683.685,Z 602.469,A 0.000,B 0.000,C 90.000,E1 300.335} C_DIS
LIN {X -0.030,Y -687.713,Z 602.462,A 0.000,B 0.000,C 90.000,E1 299.155} C_DIS
LIN {X 0.048,Y -690.041,Z 602.458,A 0.000,B 0.000,C 90.000,E1 298.437} C_DIS
LIN {X -0.226,Y -692.892,Z 602.453,A 0.000,B 0.000,C 90.000,E1 297.513} C_DIS
LIN {X -0.107,Y -694.891,Z 602.449,A 0.000,B 0.000,C 90.000,E1 296.796} C_DIS
LIN {X 0.087,Y -695.772,Z 602.446,A 0.000,B 0.000,C 90.000,E1 296.309} C_DIS
LIN {X -0.281,Y -696.105,Z 602.445,A 0.000,B 0.000,C 90.000,E1 296.104} C_DIS
LIN {X -0.026,Y -696.171,Z 602.444,A 0.000,B 0.000,C 90.000,E1 295.848} C_DIS
LIN {X -0.141,Y -695.531,Z 602.441,A 0.000,B 0.000,C 90.000,E1 295.387} C_DIS
LIN {X -0.182,Y -694.882,Z 602.440,A 0.000,B 0.000,C 90.000,E1 295.155} C_DIS
LIN {X 0.072,Y -693.408,Z 602.438,A 0.000,B 0.000,C 90.000,E1 294.899} C_DIS
LIN {X 0.258,Y -691.793,Z 602.437,A 0.000,B 0.000,C 90.000,E1 294.591} C_DIS
LIN {X -0.249,Y -690.845,Z 602.436,A 0.000,B 0.000,C 90.000,E1 294.515} C_DIS
LIN {X -0.129,Y -689.401,Z 602.435,A 0.000,B 0.000,C 90.000,E1 294.387} C_DIS
LIN {X -0.008,Y -682.682,Z 602.433,A 0.000,B 0.000,C 90.000,E1 294.003} C_DIS
LIN {X 0.222,Y -680.666,Z 602.433,A 0.000,B 0.000,C 90.000,E1 293.898} C_DIS
LIN {X 0.086,Y -676.068,Z 602.432,A 0.000,B 0.000,C 90.000,E1 293.770} C_DIS
LIN {X 0.138,Y -667.294,Z 602.431,A 0.000,B 0.000,C 90.000,E1 293.590} C_DIS
LIN {X -0.062,Y -656.867,Z 602.430,A 0.000,B 0.000,C 90.000,E1 293.462} C_DIS
LIN {X 0.041,Y -648.284,Z 602.430,A 0.000,B 0.000,C 90.000,E1 293.334} C_DIS
LIN {X 0.107,Y -638.237,Z 602.429,A 0.000,B 0.000,C 90.000,E1 293.153} C_DIS
LIN {X 0.037,Y -631.630,Z 602.428,A 0.000,B 0.000,C 90.000,E1 293.025} C_DIS
LIN {X 0.224,Y -622.073,Z 602.427,A 0.000,B 0.000,C 90.000,E1 292.770} C_DIS
LIN {X 0.036,Y -608.790,Z 602.425,A 0.000,B 0.000,C 90.000,E1 292.408} C_DIS
LIN {X 0.026,Y -581.142,Z 602.420,A 0.000,B 0.000,C 90.000,E1 291.535} C_DIS
LIN {X 0.233,Y -567.552,Z 602.417,A 0.000,B 0.000,C 90.000,E1 291.099} C_DIS
LIN {X 0.348,Y -564.487,Z 602.417,A 0.000,B 0.000,C 90.000,E1 290.972} C_DIS
LIN {X 0.101,Y -560.436,Z 602.416,A 0.000,B 0.000,C 90.000,E1 290.791} C_DIS
LIN {X 0.050,Y -560.395,Z 602.416,A 0.000,B 0.000,C 90.000,E1 290.791} C_DIS
LIN {X 0.034,Y -558.994,Z 602.415,A 0.000,B 0.000,C 90.000,E1 290.610} C_DIS
LIN {X -0.008,Y -558.977,Z 602.415,A 0.000,B 0.000,C 90.000,E1 290.610} C_DIS
LIN {X -0.176,Y -558.401,Z 602.412,A 0.000,B 0.000,C 90.000,E1 290.248} C_DIS
LIN {X 0.062,Y -558.281,Z 602.406,A 0.000,B 0.000,C 90.000,E1 289.141} C_DIS
LIN {X -0.167,Y -558.217,Z 602.400,A 0.000,B 0.000,C 90.000,E1 288.055} C_DIS
LIN {X -0.273,Y -557.899,Z 602.393,A 0.000,B 0.000,C 90.000,E1 286.677} C_DIS
LIN {X -0.130,Y -557.467,Z 602.386,A 0.000,B 0.000,C 90.000,E1 285.552} C_DIS
LIN {X 0.282,Y -556.815,Z 602.379,A 0.000,B 0.000,C 90.000,E1 284.120} C_DIS
LIN {X -0.130,Y -556.114,Z 602.371,A 0.000,B 0.000,C 90.000,E1 282.771} C_DIS
LIN {X -0.004,Y -555.297,Z 602.363,A 0.000,B 0.000,C 90.000,E1 281.366} C_DIS
LIN {X 0.102,Y -554.606,Z 602.355,A 0.000,B 0.000,C 90.000,E1 279.962} C_DIS
LIN {X 0.214,Y -553.705,Z 602.346,A 0.000,B 0.000,C 90.000,E1 278.276} C_DIS
LIN {X -0.232,Y -552.668,Z 602.334,A 0.000,B 0.000,C 90.000,E1 276.087} C_DIS
LIN {X -0.248,Y -551.902,Z 602.323,A 0.000,B 0.000,C 90.000,E1 274.131} C_DIS
LIN {X 0.229,Y -551.314,Z 602.312,A 0.000,B 0.000,C 90.000,E1 272.121} C_DIS
LIN {X -0.007,Y -550.957,Z 602.304,A 0.000,B 0.000,C 90.000,E1 270.745} C_DIS
LIN {X 0.231,Y -550.670,Z 602.298,A 0.000,B 0.000,C 90.000,E1 269.599} C_DIS
LIN {X 0.039,Y -550.043,Z 602.289,A 0.000,B 0.000,C 90.000,E1 267.936} C_DIS
LIN {X -0.168,Y -549.312,Z 602.279,A 0.000,B 0.000,C 90.000,E1 266.274} C_DIS
LIN {X 0.141,Y -548.623,Z 602.271,A 0.000,B 0.000,C 90.000,E1 264.837} C_DIS
LIN {X -0.053,Y -547.816,Z 602.264,A 0.000,B 0.000,C 90.000,E1 263.451} C_DIS
LIN {X 0.191,Y -546.850,Z 602.257,A 0.000,B 0.000,C 90.000,E1 262.299} C_DIS
LIN {X 0.044,Y -545.621,Z 602.250,A 0.000,B 0.000,C 90.000,E1 260.905} C_DIS
LIN {X 0.060,Y -543.694,Z 602.239,A 0.000,B 0.000,C 90.000,E1 258.926} C_DIS
LIN {X -0.038,Y -542.380,Z 602.231,A 0.000,B 0.000,C 90.000,E1 257.521} C_DIS
LIN {X -0.167,Y -540.979,Z 602.223,A 0.000,B 0.000,C 90.000,E1 256.117} C_DIS
LIN {X -0.061,Y -539.555,Z 602.215,A 0.000,B 0.000,C 90.000,E1 254.685} C_DIS
LIN {X 0.086,Y -537.768,Z 602.205,A 0.000,B 0.000,C 90.000,E1 252.960} C_DIS
LIN {X 0.130,Y -536.277,Z 602.198,A 0.000,B 0.000,C 90.000,E1 251.529} C_DIS
LIN {X 0.072,Y -535.316,Z 602.193,A 0.000,B 0.000,C 90.000,E1 250.678} C_DIS
LIN {X 0.005,Y -534.150,Z 602.188,A 0.000,B 0.000,C 90.000,E1 249.826} C_DIS
LIN {X 0.122,Y -532.317,Z 602.182,A 0.000,B 0.000,C 90.000,E1 248.666} C_DIS
LIN {X 0.106,Y -529.771,Z 602.174,A 0.000,B 0.000,C 90.000,E1 247.230} C_DIS
LIN {X 0.052,Y -527.030,Z 602.166,A 0.000,B 0.000,C 90.000,E1 245.793} C_DIS
LIN {X -0.223,Y -524.645,Z 602.159,A 0.000,B 0.000,C 90.000,E1 244.665} C_DIS
LIN {X 0.077,Y -521.539,Z 602.151,A 0.000,B 0.000,C 90.000,E1 243.179} C_DIS
LIN {X -0.048,Y -518.887,Z 602.145,A 0.000,B 0.000,C 90.000,E1 242.025} C_DIS
LIN {X 0.116,Y -516.803,Z 602.140,A 0.000,B 0.000,C 90.000,E1 241.129} C_DIS
LIN {X 0.066,Y -513.170,Z 602.132,A 0.000,B 0.000,C 90.000,E1 239.665} C_DIS
LIN {X -0.144,Y -508.881,Z 602.122,A 0.000,B 0.000,C 90.000,E1 237.916} C_DIS
LIN {X 0.038,Y -505.810,Z 602.115,A 0.000,B 0.000,C 90.000,E1 236.707} C_DIS
LIN {X 0.138,Y -503.323,Z 602.110,A 0.000,B 0.000,C 90.000,E1 235.801} C_DIS
LIN {X 0.094,Y -499.894,Z 602.104,A 0.000,B 0.000,C 90.000,E1 234.609} C_DIS
LIN {X -0.142,Y -491.892,Z 602.087,A 0.000,B 0.000,C 90.000,E1 231.618} C_DIS
LIN {X 0.240,Y -488.699,Z 602.080,A 0.000,B 0.000,C 90.000,E1 230.356} C_DIS
LIN {X -0.117,Y -485.598,Z 602.073,A 0.000,B 0.000,C 90.000,E1 229.175} C_DIS
LIN {X -0.018,Y -479.384,Z 602.060,A 0.000,B 0.000,C 90.000,E1 226.701} C_DIS
LIN {X 0.001,Y -474.881,Z 602.049,A 0.000,B 0.000,C 90.000,E1 224.838} C_DIS
LIN {X -0.171,Y -471.249,Z 602.040,A 0.000,B 0.000,C 90.000,E1 223.299} C_DIS
LIN {X 0.268,Y -467.683,Z 602.032,A 0.000,B 0.000,C 90.000,E1 221.676} C_DIS
LIN {X 0.131,Y -462.816,Z 602.019,A 0.000,B 0.000,C 90.000,E1 219.483} C_DIS
LIN {X -0.093,Y -458.858,Z 602.009,A 0.000,B 0.000,C 90.000,E1 217.604} C_DIS
LIN {X -0.042,Y -454.412,Z 601.996,A 0.000,B 0.000,C 90.000,E1 215.358} C_DIS
LIN {X -0.119,Y -448.934,Z 601.980,A 0.000,B 0.000,C 90.000,E1 212.467} C_DIS
LIN {X -0.062,Y -445.417,Z 601.970,A 0.000,B 0.000,C 90.000,E1 210.512} C_DIS
LIN {X 0.017,Y -442.473,Z 601.960,A 0.000,B 0.000,C 90.000,E1 208.871} C_DIS
LIN {X -0.133,Y -439.002,Z 601.950,A 0.000,B 0.000,C 90.000,E1 206.924} C_DIS
LIN {X -0.185,Y -436.126,Z 601.940,A 0.000,B 0.000,C 90.000,E1 205.283} C_DIS
LIN {X -0.112,Y -433.866,Z 601.933,A 0.000,B 0.000,C 90.000,E1 203.951} C_DIS
LIN {X 0.157,Y -430.010,Z 601.920,A 0.000,B 0.000,C 90.000,E1 201.589} C_DIS
LIN {X 0.202,Y -425.703,Z 601.905,A 0.000,B 0.000,C 90.000,E1 198.906} C_DIS
LIN {X 0.068,Y -422.221,Z 601.892,A 0.000,B 0.000,C 90.000,E1 196.567} C_DIS
LIN {X -0.092,Y -419.932,Z 601.883,A 0.000,B 0.000,C 90.000,E1 194.898} C_DIS
LIN {X -0.056,Y -417.978,Z 601.875,A 0.000,B 0.000,C 90.000,E1 193.536} C_DIS
LIN {X -0.009,Y -415.415,Z 601.866,A 0.000,B 0.000,C 90.000,E1 191.827} C_DIS
LIN {X -0.022,Y -411.227,Z 601.849,A 0.000,B 0.000,C 90.000,E1 188.746} C_DIS
LIN {X 0.076,Y -409.087,Z 601.839,A 0.000,B 0.000,C 90.000,E1 187.011} C_DIS
LIN {X 0.094,Y -406.411,Z 601.828,A 0.000,B 0.000,C 90.000,E1 184.935} C_DIS
LIN {X 0.173,Y -401.660,Z 601.802,A 0.000,B 0.000,C 90.000,E1 180.401} C_DIS
LIN {X 0.107,Y -398.966,Z 601.781,A 0.000,B 0.000,C 90.000,E1 176.560} C_DIS
LIN {X 0.133,Y -397.753,Z 601.763,A 0.000,B 0.000,C 90.000,E1 173.394} C_DIS
LIN {X -0.193,Y -397.126,Z 601.746,A 0.000,B 0.000,C 90.000,E1 170.274} C_DIS
LIN {X 0.110,Y -397.170,Z 601.728,A 0.000,B 0.000,C 90.000,E1 167.061} C_DIS
LIN {X -0.150,Y -397.681,Z 601.713,A 0.000,B 0.000,C 90.000,E1 164.283} C_DIS
LIN {X 0.170,Y -398.270,Z 601.701,A 0.000,B 0.000,C 90.000,E1 162.127} C_DIS
LIN {X -0.125,Y -398.911,Z 601.689,A 0.000,B 0.000,C 90.000,E1 160.061} C_DIS
LIN {X 0.107,Y -399.667,Z 601.677,A 0.000,B 0.000,C 90.000,E1 157.922} C_DIS
LIN {X -0.077,Y -400.550,Z 601.666,A 0.000,B 0.000,C 90.000,E1 155.845} C_DIS
LIN {X 0.060,Y -401.265,Z 601.656,A 0.000,B 0.000,C 90.000,E1 154.076} C_DIS
LIN {X -0.158,Y -402.046,Z 601.646,A 0.000,B 0.000,C 90.000,E1 152.359} C_DIS
LIN {X 0.009,Y -402.710,Z 601.637,A 0.000,B 0.000,C 90.000,E1 150.589} C_DIS
LIN {X -0.159,Y -403.338,Z 601.627,A 0.000,B 0.000,C 90.000,E1 148.869} C_DIS
LIN {X -0.009,Y -403.741,Z 601.619,A 0.000,B 0.000,C 90.000,E1 147.454} C_DIS
LIN {X -0.070,Y -404.204,Z 601.610,A 0.000,B 0.000,C 90.000,E1 145.722} C_DIS
LIN {X -0.124,Y -404.642,Z 601.600,A 0.000,B 0.000,C 90.000,E1 143.989} C_DIS
LIN {X -0.126,Y -405.255,Z 601.588,A 0.000,B 0.000,C 90.000,E1 141.904} C_DIS
LIN {X -0.007,Y -405.814,Z 601.579,A 0.000,B 0.000,C 90.000,E1 140.150} C_DIS
LIN {X 0.070,Y -406.278,Z 601.569,A 0.000,B 0.000,C 90.000,E1 138.405} C_DIS
LIN {X -0.148,Y -406.595,Z 601.559,A 0.000,B 0.000,C 90.000,E1 136.701} C_DIS
LIN {X 0.044,Y -406.916,Z 601.548,A 0.000,B 0.000,C 90.000,E1 134.595} C_DIS
LIN {X 0.120,Y -407.182,Z 601.538,A 0.000,B 0.000,C 90.000,E1 132.852} C_DIS
LIN {X 0.069,Y -407.426,Z 601.527,A 0.000,B 0.000,C 90.000,E1 130.782} C_DIS
LIN {X -0.078,Y -407.672,Z 601.517,A 0.000,B 0.000,C 90.000,E1 129.072} C_DIS
LIN {X 0.071,Y -407.712,Z 601.515,A 0.000,B 0.000,C 90.000,E1 128.705} C_DIS
LIN {X -0.099,Y -408.550,Z 601.513,A 0.000,B 0.000,C 90.000,E1 128.382} C_DIS
LIN {X -0.045,Y -415.570,Z 601.500,A 0.000,B 0.000,C 90.000,E1 125.964} C_DIS
LIN {X -0.032,Y -424.102,Z 601.481,A 0.000,B 0.000,C 90.000,E1 122.546} C_DIS
LIN {X -0.071,Y -424.159,Z 601.481,A 0.000,B 0.000,C 90.000,E1 122.546} C_DIS
LIN {X -0.223,Y -426.668,Z 601.480,A 0.000,B 0.000,C 90.000,E1 122.418} C_DIS
LIN {X 0.015,Y -443.929,Z 601.475,A 0.000,B 0.000,C 90.000,E1 121.544} C_DIS
LIN {X 0.067,Y -458.879,Z 601.471,A 0.000,B 0.000,C 90.000,E1 120.797} C_DIS
LIN {X -0.124,Y -467.185,Z 601.469,A 0.000,B 0.000,C 90.000,E1 120.384} C_DIS
LIN {X 0.150,Y -477.210,Z 601.466,A 0.000,B 0.000,C 90.000,E1 119.795} C_DIS
LIN {X -0.175,Y -483.705,Z 601.464,A 0.000,B 0.000,C 90.000,E1 119.461} C_DIS
LIN {X -0.008,Y -494.986,Z 601.460,A 0.000,B 0.000,C 90.000,E1 118.743} C_DIS
LIN {X -0.066,Y -502.837,Z 601.457,A 0.000,B 0.000,C 90.000,E1 118.231} C_DIS
LIN {X -0.068,Y -510.609,Z 601.454,A 0.000,B 0.000,C 90.000,E1 117.692} C_DIS
LIN {X -0.023,Y -518.130,Z 601.451,A 0.000,B 0.000,C 90.000,E1 117.129} C_DIS
LIN {X -0.048,Y -525.508,Z 601.448,A 0.000,B 0.000,C 90.000,E1 116.565} C_DIS
LIN {X 0.179,Y -532.514,Z 601.444,A 0.000,B 0.000,C 90.000,E1 115.976} C_DIS
LIN {X -0.094,Y -536.850,Z 601.442,A 0.000,B 0.000,C 90.000,E1 115.643} C_DIS
LIN {X -0.164,Y -542.547,Z 601.440,A 0.000,B 0.000,C 90.000,E1 115.155} C_DIS
LIN {X 0.029,Y -547.674,Z 601.437,A 0.000,B 0.000,C 90.000,E1 114.643} C_DIS
LIN {X -0.209,Y -552.284,Z 601.434,A 0.000,B 0.000,C 90.000,E1 114.207} C_DIS
LIN {X -0.062,Y -556.934,Z 601.431,A 0.000,B 0.000,C 90.000,E1 113.643} C_DIS
LIN {X -0.089,Y -562.165,Z 601.427,A 0.000,B 0.000,C 90.000,E1 112.950} C_DIS
LIN {X -0.072,Y -566.604,Z 601.424,A 0.000,B 0.000,C 90.000,E1 112.259} C_DIS
LIN {X 0.206,Y -571.192,Z 601.419,A 0.000,B 0.000,C 90.000,E1 111.408} C_DIS
LIN {X 0.091,Y -574.761,Z 601.415,A 0.000,B 0.000,C 90.000,E1 110.737} C_DIS
LIN {X 0.009,Y -577.994,Z 601.412,A 0.000,B 0.000,C 90.000,E1 110.066} C_DIS
LIN {X -0.048,Y -580.973,Z 601.408,A 0.000,B 0.000,C 90.000,E1 109.396} C_DIS
LIN {X -0.159,Y -584.273,Z 601.403,A 0.000,B 0.000,C 90.000,E1 108.598} C_DIS
LIN {X 0.130,Y -587.285,Z 601.399,A 0.000,B 0.000,C 90.000,E1 107.764} C_DIS
LIN {X 0.218,Y -589.136,Z 601.396,A 0.000,B 0.000,C 90.000,E1 107.221} C_DIS
LIN {X 0.003,Y -591.721,Z 601.391,A 0.000,B 0.000,C 90.000,E1 106.441} C_DIS
LIN {X 0.081,Y -594.859,Z 601.385,A 0.000,B 0.000,C 90.000,E1 105.371} C_DIS
LIN {X -0.061,Y -602.057,Z 601.372,A 0.000,B 0.000,C 90.000,E1 103.008} C_DIS
LIN {X -0.194,Y -607.842,Z 601.362,A 0.000,B 0.000,C 90.000,E1 101.186} C_DIS
LIN {X 0.188,Y -611.902,Z 601.355,A 0.000,B 0.000,C 90.000,E1 99.849} C_DIS
LIN {X 0.286,Y -614.999,Z 601.349,A 0.000,B 0.000,C 90.000,E1 98.803} C_DIS
LIN {X 0.058,Y -617.200,Z 601.345,A 0.000,B 0.000,C 90.000,E1 98.049} C_DIS
LIN {X -0.103,Y -620.719,Z 601.338,A 0.000,B 0.000,C 90.000,E1 96.777} C_DIS
LIN {X 0.027,Y -623.383,Z 601.332,A 0.000,B 0.000,C 90.000,E1 95.739} C_DIS
LIN {X 0.188,Y -625.717,Z 601.326,A 0.000,B 0.000,C 90.000,E1 94.702} C_DIS
LIN {X -0.012,Y -627.240,Z 601.322,A 0.000,B 0.000,C 90.000,E1 93.955} C_DIS
LIN {X 0.150,Y -629.072,Z 601.316,A 0.000,B 0.000,C 90.000,E1 92.922} C_DIS
LIN {X 0.063,Y -630.987,Z 601.309,A 0.000,B 0.000,C 90.000,E1 91.661} C_DIS
LIN {X -0.110,Y -631.935,Z 601.305,A 0.000,B 0.000,C 90.000,E1 90.917} C_DIS
LIN {X -0.270,Y -632.693,Z 601.301,A 0.000,B 0.000,C 90.000,E1 90.172} C_DIS
LIN {X 0.210,Y -633.206,Z 601.297,A 0.000,B 0.000,C 90.000,E1 89.370} C_DIS
LIN {X 0.061,Y -633.495,Z 601.292,A 0.000,B 0.000,C 90.000,E1 88.625} C_DIS
LIN {X -0.068,Y -633.657,Z 601.288,A 0.000,B 0.000,C 90.000,E1 87.879} C_DIS
LIN {X -0.077,Y -633.310,Z 601.281,A 0.000,B 0.000,C 90.000,E1 86.617} C_DIS
LIN {X 0.168,Y -632.751,Z 601.276,A 0.000,B 0.000,C 90.000,E1 85.584} C_DIS
LIN {X 0.181,Y -631.670,Z 601.269,A 0.000,B 0.000,C 90.000,E1 84.318} C_DIS
LIN {X 0.039,Y -630.887,Z 601.264,A 0.000,B 0.000,C 90.000,E1 83.571} C_DIS
LIN {X -0.039,Y -629.909,Z 601.260,A 0.000,B 0.000,C 90.000,E1 82.818} C_DIS
LIN {X 0.204,Y -628.249,Z 601.255,A 0.000,B 0.000,C 90.000,E1 81.781} C_DIS
LIN {X -0.107,Y -626.379,Z 601.249,A 0.000,B 0.000,C 90.000,E1 80.792} C_DIS
LIN {X 0.178,Y -624.300,Z 601.243,A 0.000,B 0.000,C 90.000,E1 79.746} C_DIS
LIN {X 0.209,Y -621.412,Z 601.236,A 0.000,B 0.000,C 90.000,E1 78.465} C_DIS
LIN {X 0.315,Y -618.259,Z 601.229,A 0.000,B 0.000,C 90.000,E1 77.173} C_DIS
LIN {X 0.233,Y -616.200,Z 601.225,A 0.000,B 0.000,C 90.000,E1 76.408} C_DIS
LIN {X -0.350,Y -612.546,Z 601.217,A 0.000,B 0.000,C 90.000,E1 75.172} C_DIS
LIN {X 0.254,Y -610.211,Z 601.213,A 0.000,B 0.000,C 90.000,E1 74.338} C_DIS
LIN {X -0.080,Y -608.529,Z 601.210,A 0.000,B 0.000,C 90.000,E1 73.850} C_DIS
LIN {X -0.010,Y -606.802,Z 601.207,A 0.000,B 0.000,C 90.000,E1 73.323} C_DIS
LIN {X -0.047,Y -603.951,Z 601.203,A 0.000,B 0.000,C 90.000,E1 72.543} C_DIS
LIN {X -0.115,Y -600.781,Z 601.199,A 0.000,B 0.000,C 90.000,E1 71.764} C_DIS
LIN {X -0.025,Y -597.349,Z 601.194,A 0.000,B 0.000,C 90.000,E1 70.967} C_DIS
LIN {X -0.220,Y -593.004,Z 601.189,A 0.000,B 0.000,C 90.000,E1 70.061} C_DIS
LIN {X 0.283,Y -588.387,Z 601.184,A 0.000,B 0.000,C 90.000,E1 69.082} C_DIS
LIN {X 0.243,Y -583.991,Z 601.180,A 0.000,B 0.000,C 90.000,E1 68.284} C_DIS
LIN {X -0.311,Y -580.058,Z 601.176,A 0.000,B 0.000,C 90.000,E1 67.667} C_DIS
LIN {X -0.137,Y -575.703,Z 601.172,A 0.000,B 0.000,C 90.000,E1 66.975} C_DIS
LIN {X -0.230,Y -570.786,Z 601.168,A 0.000,B 0.000,C 90.000,E1 66.305} C_DIS
LIN {X -0.052,Y -566.513,Z 601.165,A 0.000,B 0.000,C 90.000,E1 65.741} C_DIS
LIN {X 0.093,Y -561.899,Z 601.162,A 0.000,B 0.000,C 90.000,E1 65.177} C_DIS
LIN {X 0.058,Y -555.942,Z 601.159,A 0.000,B 0.000,C 90.000,E1 64.537} C_DIS
LIN {X 0.219,Y -550.850,Z 601.156,A 0.000,B 0.000,C 90.000,E1 64.024} C_DIS
LIN {X -0.137,Y -545.366,Z 601.153,A 0.000,B 0.000,C 90.000,E1 63.589} C_DIS
LIN {X 0.005,Y -542.321,Z 601.152,A 0.000,B 0.000,C 90.000,E1 63.332} C_DIS
LIN {X -0.054,Y -536.303,Z 601.150,A 0.000,B 0.000,C 90.000,E1 62.922} C_DIS
LIN {X 0.171,Y -529.602,Z 601.147,A 0.000,B 0.000,C 90.000,E1 62.487} C_DIS
LIN {X -0.087,Y -519.551,Z 601.144,A 0.000,B 0.000,C 90.000,E1 61.975} C_DIS
LIN {X -0.172,Y -510.885,Z 601.142,A 0.000,B 0.000,C 90.000,E1 61.563} C_DIS
LIN {X 0.149,Y -502.243,Z 601.140,A 0.000,B 0.000,C 90.000,E1 61.129} C_DIS
LIN {X -0.087,Y -485.238,Z 601.135,A 0.000,B 0.000,C 90.000,E1 60.383} C_DIS
LIN {X -0.184,Y -476.656,Z 601.133,A 0.000,B 0.000,C 90.000,E1 59.999} C_DIS
LIN {X 0.176,Y -463.414,Z 601.130,A 0.000,B 0.000,C 90.000,E1 59.331} C_DIS
LIN {X 0.146,Y -447.862,Z 601.125,A 0.000,B 0.000,C 90.000,E1 58.535} C_DIS
LIN {X 0.103,Y -447.796,Z 601.125,A 0.000,B 0.000,C 90.000,E1 58.535} C_DIS
LIN {X 0.173,Y -443.835,Z 601.114,A 0.000,B 0.000,C 90.000,E1 56.421} C_DIS
LIN {X 0.185,Y -434.687,Z 601.092,A 0.000,B 0.000,C 90.000,E1 52.477} C_DIS
LIN {X -0.038,Y -431.562,Z 601.083,A 0.000,B 0.000,C 90.000,E1 50.848} C_DIS
LIN {X -0.015,Y -431.558,Z 601.082,A 0.000,B 0.000,C 90.000,E1 50.678} C_DIS
LIN {X -0.229,Y -432.438,Z 601.075,A 0.000,B 0.000,C 90.000,E1 49.542} C_DIS
LIN {X 0.084,Y -433.558,Z 601.066,A 0.000,B 0.000,C 90.000,E1 47.838} C_DIS
LIN {X -0.135,Y -434.468,Z 601.059,A 0.000,B 0.000,C 90.000,E1 46.539} C_DIS
LIN {X 0.101,Y -436.038,Z 601.046,A 0.000,B 0.000,C 90.000,E1 44.190} C_DIS
LIN {X 0.218,Y -436.935,Z 601.038,A 0.000,B 0.000,C 90.000,E1 42.852} C_DIS
LIN {X 0.056,Y -437.698,Z 601.031,A 0.000,B 0.000,C 90.000,E1 41.553} C_DIS
LIN {X -0.145,Y -438.519,Z 601.022,A 0.000,B 0.000,C 90.000,E1 39.930} C_DIS
LIN {X 0.003,Y -439.349,Z 601.011,A 0.000,B 0.000,C 90.000,E1 37.935} C_DIS
LIN {X -0.015,Y -439.922,Z 601.000,A 0.000,B 0.000,C 90.000,E1 35.964} C_DIS
LIN {X -0.051,Y -440.218,Z 600.991,A 0.000,B 0.000,C 90.000,E1 34.326} C_DIS
LIN {X -0.016,Y -440.447,Z 600.983,A 0.000,B 0.000,C 90.000,E1 33.007} C_DIS
LIN {X 0.155,Y -440.578,Z 600.976,A 0.000,B 0.000,C 90.000,E1 31.671} C_DIS
LIN {X -0.134,Y -440.922,Z 600.963,A 0.000,B 0.000,C 90.000,E1 29.411} C_DIS
LIN {X 0.144,Y -441.215,Z 600.951,A 0.000,B 0.000,C 90.000,E1 27.078} C_DIS
LIN {X -0.052,Y -441.494,Z 600.941,A 0.000,B 0.000,C 90.000,E1 25.463} C_DIS
LIN {X -0.192,Y -441.924,Z 600.931,A 0.000,B 0.000,C 90.000,E1 23.515} C_DIS
LIN {X 0.059,Y -442.342,Z 600.921,A 0.000,B 0.000,C 90.000,E1 21.844} C_DIS
LIN {X 0.018,Y -442.890,Z 600.911,A 0.000,B 0.000,C 90.000,E1 19.885} C_DIS
LIN {X -0.160,Y -443.532,Z 600.900,A 0.000,B 0.000,C 90.000,E1 17.946} C_DIS
LIN {X 0.085,Y -444.510,Z 600.885,A 0.000,B 0.000,C 90.000,E1 15.300} C_DIS
LIN {X -0.006,Y -445.780,Z 600.871,A 0.000,B 0.000,C 90.000,E1 12.703} C_DIS
LIN {X -0.147,Y -447.650,Z 600.854,A 0.000,B 0.000,C 90.000,E1 9.792} C_DIS
LIN {X -0.035,Y -449.582,Z 600.840,A 0.000,B 0.000,C 90.000,E1 7.182} C_DIS
LIN {X 0.121,Y -451.222,Z 600.829,A 0.000,B 0.000,C 90.000,E1 5.220} C_DIS
LIN {X 0.075,Y -452.799,Z 600.820,A 0.000,B 0.000,C 90.000,E1 3.612} C_DIS
LIN {X -0.051,Y -455.201,Z 600.808,A 0.000,B 0.000,C 90.000,E1 1.375} C_DIS
LIN {X 0.015,Y -458.792,Z 600.792,A 0.000,B 0.000,C 90.000,E1 358.511} C_DIS
LIN {X -0.228,Y -463.457,Z 600.774,A 0.000,B 0.000,C 90.000,E1 355.355} C_DIS
LIN {X -0.197,Y -466.412,Z 600.764,A 0.000,B 0.000,C 90.000,E1 353.451} C_DIS
LIN {X 0.100,Y -468.954,Z 600.755,A 0.000,B 0.000,C 90.000,E1 351.837} C_DIS
LIN {X -0.142,Y -471.864,Z 600.744,A 0.000,B 0.000,C 90.000,E1 349.982} C_DIS
LIN {X 0.158,Y -475.391,Z 600.732,A 0.000,B 0.000,C 90.000,E1 347.757} C_DIS
LIN {X 0.091,Y -477.591,Z 600.725,A 0.000,B 0.000,C 90.000,E1 346.520} C_DIS
LIN {X -0.121,Y -480.945,Z 600.715,A 0.000,B 0.000,C 90.000,E1 344.685} C_DIS
LIN {X -0.126,Y -483.798,Z 600.706,A 0.000,B 0.000,C 90.000,E1 343.142} C_DIS
LIN {X 0.066,Y -487.305,Z 600.696,A 0.000,B 0.000,C 90.000,E1 341.275} C_DIS
LIN {X -0.017,Y -489.702,Z 600.689,A 0.000,B 0.000,C 90.000,E1 340.061} C_DIS
LIN {X -0.033,Y -492.603,Z 600.681,A 0.000,B 0.000,C 90.000,E1 338.539} C_DIS
LIN {X -0.279,Y -495.309,Z 600.672,A 0.000,B 0.000,C 90.000,E1 337.050} C_DIS
LIN {X 0.178,Y -497.830,Z 600.664,A 0.000,B 0.000,C 90.000,E1 335.485} C_DIS
LIN {X 0.060,Y -500.647,Z 600.654,A 0.000,B 0.000,C 90.000,E1 333.691} C_DIS
LIN {X 0.090,Y -502.456,Z 600.647,A 0.000,B 0.000,C 90.000,E1 332.487} C_DIS
LIN {X -0.137,Y -505.158,Z 600.637,A 0.000,B 0.000,C 90.000,E1 330.717} C_DIS
LIN {X 0.014,Y -508.280,Z 600.626,A 0.000,B 0.000,C 90.000,E1 328.614} C_DIS
LIN {X -0.087,Y -511.742,Z 600.614,A 0.000,B 0.000,C 90.000,E1 326.548} C_DIS
LIN {X -0.162,Y -516.231,Z 600.601,A 0.000,B 0.000,C 90.000,E1 324.196} C_DIS
LIN {X -0.070,Y -519.145,Z 600.593,A 0.000,B 0.000,C 90.000,E1 322.718} C_DIS
LIN {X -0.074,Y -522.801,Z 600.583,A 0.000,B 0.000,C 90.000,E1 320.964} C_DIS
LIN {X 0.121,Y -525.313,Z 600.578,A 0.000,B 0.000,C 90.000,E1 320.070} C_DIS
LIN {X -0.171,Y -526.881,Z 600.576,A 0.000,B 0.000,C 90.000,E1 319.666} C_DIS
LIN {X -0.195,Y -530.726,Z 600.572,A 0.000,B 0.000,C 90.000,E1 318.933} C_DIS
LIN {X -0.034,Y -531.736,Z 600.571,A 0.000,B 0.000,C 90.000,E1 318.771} C_DIS
LIN {X 0.191,Y -535.912,Z 600.569,A 0.000,B 0.000,C 90.000,E1 318.324} C_DIS
LIN {X -0.320,Y -537.089,Z 600.568,A 0.000,B 0.000,C 90.000,E1 318.243} C_DIS
LIN {X -0.012,Y -541.904,Z 600.565,A 0.000,B 0.000,C 90.000,E1 317.757} C_DIS
LIN {X 0.194,Y -558.130,Z 600.558,A 0.000,B 0.000,C 90.000,E1 316.458} C_DIS
LIN {X -0.229,Y -571.432,Z 600.553,A 0.000,B 0.000,C 90.000,E1 315.486} C_DIS
LIN {X -0.049,Y -583.222,Z 600.548,A 0.000,B 0.000,C 90.000,E1 314.595} C_DIS
LIN {X 0.166,Y -590.436,Z 600.545,A 0.000,B 0.000,C 90.000,E1 314.028} C_DIS
LIN {X -0.119,Y -598.870,Z 600.541,A 0.000,B 0.000,C 90.000,E1 313.380} C_DIS
LIN {X -0.297,Y -604.285,Z 600.538,A 0.000,B 0.000,C 90.000,E1 312.933} C_DIS
LIN {X -0.245,Y -609.411,Z 600.536,A 0.000,B 0.000,C 90.000,E1 312.447} C_DIS
LIN {X 0.080,Y -617.940,Z 600.531,A 0.000,B 0.000,C 90.000,E1 311.553} C_DIS
LIN {X -0.191,Y -622.558,Z 600.528,A 0.000,B 0.000,C 90.000,E1 311.067} C_DIS
LIN {X -0.022,Y -632.057,Z 600.522,A 0.000,B 0.000,C 90.000,E1 309.930} C_DIS
LIN {X -0.296,Y -638.287,Z 600.518,A 0.000,B 0.000,C 90.000,E1 309.197} C_DIS
LIN {X -0.107,Y -645.088,Z 600.513,A 0.000,B 0.000,C 90.000,E1 308.302} C_DIS
LIN {X -0.175,Y -648.743,Z 600.510,A 0.000,B 0.000,C 90.000,E1 307.810} C_DIS
LIN {X -0.293,Y -653.700,Z 600.506,A 0.000,B 0.000,C 90.000,E1 307.076} C_DIS
LIN {X 0.191,Y -656.015,Z 600.504,A 0.000,B 0.000,C 90.000,E1 306.664} C_DIS
LIN {X 0.141,Y -660.124,Z 600.500,A 0.000,B 0.000,C 90.000,E1 305.931} C_DIS
LIN {X 0.178,Y -662.624,Z 600.497,A 0.000,B 0.000,C 90.000,E1 305.438} C_DIS
LIN {X 0.228,Y -665.007,Z 600.494,A 0.000,B 0.000,C 90.000,E1 304.945} C_DIS
LIN {X -0.005,Y -669.223,Z 600.489,A 0.000,B 0.000,C 90.000,E1 303.992} C_DIS
LIN {X -0.329,Y -672.120,Z 600.485,A 0.000,B 0.000,C 90.000,E1 303.293} C_DIS
LIN {X 0.227,Y -677.478,Z 600.477,A 0.000,B 0.000,C 90.000,E1 301.799} C_DIS
LIN {X -0.049,Y -682.595,Z 600.469,A 0.000,B 0.000,C 90.000,E1 300.384} C_DIS
LIN {X 0.182,Y -685.866,Z 600.464,A 0.000,B 0.000,C 90.000,E1 299.411} C_DIS
LIN {X -0.139,Y -688.987,Z 600.458,A 0.000,B 0.000,C 90.000,E1 298.487} C_DIS
LIN {X 0.183,Y -691.934,Z 600.453,A 0.000,B 0.000,C 90.000,E1 297.513} C_DIS
LIN {X -0.019,Y -693.980,Z 600.449,A 0.000,B 0.000,C 90.000,E1 296.821} C_DIS
LIN {X -0.391,Y -694.505,Z 600.448,A 0.000,B 0.000,C 90.000,E1 296.616} C_DIS
LIN {X 0.112,Y -695.271,Z 600.445,A 0.000,B 0.000,C 90.000,E1 296.104} C_DIS
LIN {X 0.364,Y -695.355,Z 600.444,A 0.000,B 0.000,C 90.000,E1 295.848} C_DIS
LIN {X -0.054,Y -694.760,Z 600.441,A 0.000,B 0.000,C 90.000,E1 295.412} C_DIS
LIN {X 0.199,Y -694.130,Z 600.440,A 0.000,B 0.000,C 90.000,E1 295.155} C_DIS
LIN {X 0.067,Y -691.561,Z 600.437,A 0.000,B 0.000,C 90.000,E1 294.695} C_DIS
LIN {X -0.100,Y -690.803,Z 600.437,A 0.000,B 0.000,C 90.000,E1 294.591} C_DIS
LIN {X 0.020,Y -689.649,Z 600.436,A 0.000,B 0.000,C 90.000,E1 294.463} C_DIS
LIN {X 0.139,Y -687.845,Z 600.435,A 0.000,B 0.000,C 90.000,E1 294.335} C_DIS
LIN {X -0.250,Y -682.765,Z 600.434,A 0.000,B 0.000,C 90.000,E1 294.079} C_DIS
LIN {X -0.265,Y -679.907,Z 600.433,A 0.000,B 0.000,C 90.000,E1 293.951} C_DIS
LIN {X 0.130,Y -675.110,Z 600.432,A 0.000,B 0.000,C 90.000,E1 293.770} C_DIS
LIN {X -0.016,Y -668.754,Z 600.431,A 0.000,B 0.000,C 90.000,E1 293.643} C_DIS
LIN {X -0.225,Y -659.380,Z 600.431,A 0.000,B 0.000,C 90.000,E1 293.515} C_DIS
LIN {X 0.116,Y -648.127,Z 600.430,A 0.000,B 0.000,C 90.000,E1 293.334} C_DIS
LIN {X -0.372,Y -638.302,Z 600.429,A 0.000,B 0.000,C 90.000,E1 293.206} C_DIS
LIN {X 0.190,Y -628.733,Z 600.428,A 0.000,B 0.000,C 90.000,E1 292.950} C_DIS
LIN {X -0.024,Y -618.965,Z 600.426,A 0.000,B 0.000,C 90.000,E1 292.717} C_DIS
LIN {X 0.271,Y -598.671,Z 600.423,A 0.000,B 0.000,C 90.000,E1 292.078} C_DIS
LIN {X 0.285,Y -577.633,Z 600.419,A 0.000,B 0.000,C 90.000,E1 291.408} C_DIS
LIN {X -0.198,Y -567.776,Z 600.417,A 0.000,B 0.000,C 90.000,E1 291.153} C_DIS
LIN {X -0.282,Y -564.635,Z 600.417,A 0.000,B 0.000,C 90.000,E1 291.046} C_DIS
LIN {X 0.118,Y -560.557,Z 600.416,A 0.000,B 0.000,C 90.000,E1 290.791} C_DIS
LIN {X 0.067,Y -560.506,Z 600.416,A 0.000,B 0.000,C 90.000,E1 290.791} C_DIS
LIN {X 0.068,Y -559.220,Z 600.415,A 0.000,B 0.000,C 90.000,E1 290.610} C_DIS
LIN {X 0.026,Y -559.196,Z 600.415,A 0.000,B 0.000,C 90.000,E1 290.610} C_DIS
LIN {X -0.242,Y -558.636,Z 600.412,A 0.000,B 0.000,C 90.000,E1 290.248} C_DIS
LIN {X -0.185,Y -558.512,Z 600.407,A 0.000,B 0.000,C 90.000,E1 289.214} C_DIS
LIN {X -0.108,Y -558.403,Z 600.399,A 0.000,B 0.000,C 90.000,E1 287.819} C_DIS
LIN {X -0.206,Y -558.014,Z 600.391,A 0.000,B 0.000,C 90.000,E1 286.441} C_DIS
LIN {X 0.219,Y -557.460,Z 600.384,A 0.000,B 0.000,C 90.000,E1 285.009} C_DIS
LIN {X 0.081,Y -556.620,Z 600.374,A 0.000,B 0.000,C 90.000,E1 283.355} C_DIS
LIN {X 0.212,Y -555.857,Z 600.367,A 0.000,B 0.000,C 90.000,E1 281.951} C_DIS
LIN {X 0.043,Y -554.793,Z 600.356,A 0.000,B 0.000,C 90.000,E1 280.018} C_DIS
LIN {X 0.197,Y -553.743,Z 600.345,A 0.000,B 0.000,C 90.000,E1 278.049} C_DIS
LIN {X 0.210,Y -552.974,Z 600.336,A 0.000,B 0.000,C 90.000,E1 276.372} C_DIS
LIN {X 0.193,Y -552.182,Z 600.325,A 0.000,B 0.000,C 90.000,E1 274.416} C_DIS
LIN {X 0.120,Y -551.551,Z 600.314,A 0.000,B 0.000,C 90.000,E1 272.465} C_DIS
LIN {X -0.114,Y -551.216,Z 600.306,A 0.000,B 0.000,C 90.000,E1 271.088} C_DIS
LIN {X 0.186,Y -550.847,Z 600.298,A 0.000,B 0.000,C 90.000,E1 269.656} C_DIS
LIN {X 0.055,Y -550.087,Z 600.287,A 0.000,B 0.000,C 90.000,E1 267.707} C_DIS
LIN {X -0.203,Y -549.522,Z 600.280,A 0.000,B 0.000,C 90.000,E1 266.331} C_DIS
LIN {X 0.111,Y -548.835,Z 600.272,A 0.000,B 0.000,C 90.000,E1 264.894} C_DIS
LIN {X -0.140,Y -548.032,Z 600.264,A 0.000,B 0.000,C 90.000,E1 263.514} C_DIS
LIN {X 0.171,Y -547.085,Z 600.258,A 0.000,B 0.000,C 90.000,E1 262.356} C_DIS
LIN {X -0.055,Y -545.851,Z 600.250,A 0.000,B 0.000,C 90.000,E1 260.971} C_DIS
LIN {X -0.049,Y -543.926,Z 600.239,A 0.000,B 0.000,C 90.000,E1 258.993} C_DIS
LIN {X -0.236,Y -542.879,Z 600.233,A 0.000,B 0.000,C 90.000,E1 257.881} C_DIS
LIN {X -0.236,Y -541.473,Z 600.225,A 0.000,B 0.000,C 90.000,E1 256.464} C_DIS
LIN {X -0.254,Y -540.058,Z 600.217,A 0.000,B 0.000,C 90.000,E1 255.046} C_DIS
LIN {X -0.099,Y -538.300,Z 600.207,A 0.000,B 0.000,C 90.000,E1 253.323} C_DIS
LIN {X 0.123,Y -536.812,Z 600.199,A 0.000,B 0.000,C 90.000,E1 251.873} C_DIS
LIN {X -0.097,Y -535.914,Z 600.195,A 0.000,B 0.000,C 90.000,E1 251.040} C_DIS
LIN {X 0.254,Y -533.968,Z 600.187,A 0.000,B 0.000,C 90.000,E1 249.571} C_DIS
LIN {X 0.075,Y -531.529,Z 600.179,A 0.000,B 0.000,C 90.000,E1 248.156} C_DIS
LIN {X 0.147,Y -529.407,Z 600.172,A 0.000,B 0.000,C 90.000,E1 246.997} C_DIS
LIN {X 0.295,Y -526.612,Z 600.164,A 0.000,B 0.000,C 90.000,E1 245.537} C_DIS
LIN {X 0.015,Y -524.229,Z 600.158,A 0.000,B 0.000,C 90.000,E1 244.409} C_DIS
LIN {X 0.070,Y -521.074,Z 600.150,A 0.000,B 0.000,C 90.000,E1 242.948} C_DIS
LIN {X -0.158,Y -517.744,Z 600.142,A 0.000,B 0.000,C 90.000,E1 241.513} C_DIS
LIN {X 0.259,Y -514.089,Z 600.134,A 0.000,B 0.000,C 90.000,E1 239.999} C_DIS
LIN {X -0.298,Y -509.028,Z 600.122,A 0.000,B 0.000,C 90.000,E1 237.995} C_DIS
LIN {X -0.115,Y -505.994,Z 600.115,A 0.000,B 0.000,C 90.000,E1 236.786} C_DIS
LIN {X -0.015,Y -503.498,Z 600.110,A 0.000,B 0.000,C 90.000,E1 235.881} C_DIS
LIN {X -0.178,Y -499.195,Z 600.102,A 0.000,B 0.000,C 90.000,E1 234.402} C_DIS
LIN {X 0.012,Y -491.993,Z 600.087,A 0.000,B 0.000,C 90.000,E1 231.662} C_DIS
LIN {X 0.090,Y -488.801,Z 600.080,A 0.000,B 0.000,C 90.000,E1 230.436} C_DIS
LIN {X 0.052,Y -485.679,Z 600.074,A 0.000,B 0.000,C 90.000,E1 229.218} C_DIS
LIN {X -0.164,Y -479.461,Z 600.060,A 0.000,B 0.000,C 90.000,E1 226.782} C_DIS
LIN {X -0.142,Y -474.958,Z 600.049,A 0.000,B 0.000,C 90.000,E1 224.919} C_DIS
LIN {X 0.030,Y -471.331,Z 600.041,A 0.000,B 0.000,C 90.000,E1 223.338} C_DIS
LIN {X 0.130,Y -467.730,Z 600.032,A 0.000,B 0.000,C 90.000,E1 221.757} C_DIS
LIN {X -0.052,Y -463.529,Z 600.022,A 0.000,B 0.000,C 90.000,E1 219.886} C_DIS
LIN {X 0.035,Y -459.554,Z 600.011,A 0.000,B 0.000,C 90.000,E1 217.971} C_DIS
LIN {X 0.109,Y -455.080,Z 599.999,A 0.000,B 0.000,C 90.000,E1 215.724} C_DIS
LIN {X -0.106,Y -450.692,Z 599.986,A 0.000,B 0.000,C 90.000,E1 213.499} C_DIS
LIN {X -0.075,Y -447.718,Z 599.977,A 0.000,B 0.000,C 90.000,E1 211.878} C_DIS
LIN {X -0.169,Y -445.439,Z 599.970,A 0.000,B 0.000,C 90.000,E1 210.590} C_DIS
LIN {X -0.033,Y -441.894,Z 599.959,A 0.000,B 0.000,C 90.000,E1 208.615} C_DIS
LIN {X 0.198,Y -438.438,Z 599.948,A 0.000,B 0.000,C 90.000,E1 206.616} C_DIS
LIN {X -0.257,Y -435.572,Z 599.939,A 0.000,B 0.000,C 90.000,E1 205.027} C_DIS
LIN {X -0.152,Y -432.176,Z 599.928,A 0.000,B 0.000,C 90.000,E1 203.025} C_DIS
LIN {X -0.102,Y -429.471,Z 599.919,A 0.000,B 0.000,C 90.000,E1 201.354} C_DIS
LIN {X -0.122,Y -425.731,Z 599.906,A 0.000,B 0.000,C 90.000,E1 199.014} C_DIS
LIN {X -0.042,Y -422.770,Z 599.894,A 0.000,B 0.000,C 90.000,E1 196.985} C_DIS
LIN {X -0.022,Y -419.983,Z 599.883,A 0.000,B 0.000,C 90.000,E1 194.954} C_DIS
LIN {X 0.013,Y -418.066,Z 599.876,A 0.000,B 0.000,C 90.000,E1 193.592} C_DIS
LIN {X -0.080,Y -416.040,Z 599.868,A 0.000,B 0.000,C 90.000,E1 192.243} C_DIS
LIN {X 0.008,Y -411.750,Z 599.851,A 0.000,B 0.000,C 90.000,E1 189.151} C_DIS
LIN {X 0.142,Y -409.212,Z 599.839,A 0.000,B 0.000,C 90.000,E1 187.068} C_DIS
LIN {X 0.188,Y -406.959,Z 599.830,A 0.000,B 0.000,C 90.000,E1 185.334} C_DIS
LIN {X -0.157,Y -401.781,Z 599.803,A 0.000,B 0.000,C 90.000,E1 180.516} C_DIS
LIN {X -0.185,Y -399.285,Z 599.783,A 0.000,B 0.000,C 90.000,E1 177.020} C_DIS
LIN {X 0.171,Y -397.853,Z 599.764,A 0.000,B 0.000,C 90.000,E1 173.457} C_DIS
LIN {X -0.078,Y -397.275,Z 599.748,A 0.000,B 0.000,C 90.000,E1 170.679} C_DIS
LIN {X -0.151,Y -397.222,Z 599.731,A 0.000,B 0.000,C 90.000,E1 167.521} C_DIS
LIN {X -0.078,Y -397.595,Z 599.717,A 0.000,B 0.000,C 90.000,E1 165.046} C_DIS
LIN {X -0.174,Y -398.266,Z 599.703,A 0.000,B 0.000,C 90.000,E1 162.598} C_DIS
LIN {X 0.136,Y -398.685,Z 599.695,A 0.000,B 0.000,C 90.000,E1 161.148} C_DIS
LIN {X -0.144,Y -399.416,Z 599.684,A 0.000,B 0.000,C 90.000,E1 159.082} C_DIS
LIN {X -0.121,Y -400.244,Z 599.672,A 0.000,B 0.000,C 90.000,E1 156.975} C_DIS
LIN {X 0.082,Y -401.152,Z 599.660,A 0.000,B 0.000,C 90.000,E1 154.845} C_DIS
LIN {X -0.002,Y -402.228,Z 599.647,A 0.000,B 0.000,C 90.000,E1 152.410} C_DIS
LIN {X 0.084,Y -402.780,Z 599.639,A 0.000,B 0.000,C 90.000,E1 151.001} C_DIS
LIN {X -0.088,Y -403.429,Z 599.629,A 0.000,B 0.000,C 90.000,E1 149.282} C_DIS
LIN {X -0.040,Y -403.965,Z 599.620,A 0.000,B 0.000,C 90.000,E1 147.533} C_DIS
LIN {X -0.101,Y -404.393,Z 599.610,A 0.000,B 0.000,C 90.000,E1 145.801} C_DIS
LIN {X -0.152,Y -404.830,Z 599.600,A 0.000,B 0.000,C 90.000,E1 144.069} C_DIS
LIN {X -0.043,Y -405.325,Z 599.591,A 0.000,B 0.000,C 90.000,E1 142.316} C_DIS
LIN {X -0.033,Y -405.969,Z 599.579,A 0.000,B 0.000,C 90.000,E1 140.231} C_DIS
LIN {X 0.045,Y -406.424,Z 599.569,A 0.000,B 0.000,C 90.000,E1 138.485} C_DIS
LIN {X 0.108,Y -406.745,Z 599.560,A 0.000,B 0.000,C 90.000,E1 136.743} C_DIS
LIN {X 0.024,Y -407.059,Z 599.548,A 0.000,B 0.000,C 90.000,E1 134.676} C_DIS
LIN {X 0.105,Y -407.305,Z 599.539,A 0.000,B 0.000,C 90.000,E1 132.933} C_DIS
LIN {X 0.057,Y -407.517,Z 599.527,A 0.000,B 0.000,C 90.000,E1 130.862} C_DIS
LIN {X 0.170,Y -407.746,Z 599.518,A 0.000,B 0.000,C 90.000,E1 129.116} C_DIS
LIN {X -0.032,Y -407.757,Z 599.515,A 0.000,B 0.000,C 90.000,E1 128.669} C_DIS
LIN {X 0.187,Y -415.331,Z 599.500,A 0.000,B 0.000,C 90.000,E1 126.011} C_DIS
LIN {X 0.031,Y -419.417,Z 599.491,A 0.000,B 0.000,C 90.000,E1 124.326} C_DIS
LIN {X -0.118,Y -424.931,Z 599.479,A 0.000,B 0.000,C 90.000,E1 122.260} C_DIS
LIN {X 0.203,Y -425.014,Z 599.479,A 0.000,B 0.000,C 90.000,E1 122.212} C_DIS
LIN {X -0.121,Y -435.816,Z 599.476,A 0.000,B 0.000,C 90.000,E1 121.720} C_DIS
LIN {X 0.050,Y -440.970,Z 599.475,A 0.000,B 0.000,C 90.000,E1 121.465} C_DIS
LIN {X 0.202,Y -454.218,Z 599.471,A 0.000,B 0.000,C 90.000,E1 120.797} C_DIS
LIN {X 0.161,Y -467.325,Z 599.468,A 0.000,B 0.000,C 90.000,E1 120.129} C_DIS
LIN {X -0.060,Y -477.135,Z 599.465,A 0.000,B 0.000,C 90.000,E1 119.617} C_DIS
LIN {X 0.289,Y -483.707,Z 599.462,A 0.000,B 0.000,C 90.000,E1 119.205} C_DIS
LIN {X -0.153,Y -495.034,Z 599.459,A 0.000,B 0.000,C 90.000,E1 118.565} C_DIS
LIN {X -0.139,Y -501.326,Z 599.456,A 0.000,B 0.000,C 90.000,E1 118.153} C_DIS
LIN {X -0.132,Y -510.739,Z 599.453,A 0.000,B 0.000,C 90.000,E1 117.513} C_DIS
LIN {X 0.099,Y -519.798,Z 599.449,A 0.000,B 0.000,C 90.000,E1 116.821} C_DIS
LIN {X 0.273,Y -527.219,Z 599.446,A 0.000,B 0.000,C 90.000,E1 116.232} C_DIS
LIN {X 0.079,Y -534.438,Z 599.443,A 0.000,B 0.000,C 90.000,E1 115.668} C_DIS
LIN {X 0.043,Y -541.572,Z 599.439,A 0.000,B 0.000,C 90.000,E1 115.079} C_DIS
LIN {X -0.059,Y -548.197,Z 599.436,A 0.000,B 0.000,C 90.000,E1 114.463} C_DIS
LIN {X -0.106,Y -552.146,Z 599.434,A 0.000,B 0.000,C 90.000,E1 114.079} C_DIS
LIN {X 0.046,Y -556.880,Z 599.431,A 0.000,B 0.000,C 90.000,E1 113.515} C_DIS
LIN {X 0.124,Y -561.196,Z 599.428,A 0.000,B 0.000,C 90.000,E1 112.950} C_DIS
LIN {X -0.013,Y -566.307,Z 599.423,A 0.000,B 0.000,C 90.000,E1 112.206} C_DIS
LIN {X 0.102,Y -570.172,Z 599.420,A 0.000,B 0.000,C 90.000,E1 111.535} C_DIS
LIN {X -0.109,Y -574.537,Z 599.415,A 0.000,B 0.000,C 90.000,E1 110.737} C_DIS
LIN {X -0.195,Y -577.863,Z 599.411,A 0.000,B 0.000,C 90.000,E1 110.066} C_DIS
LIN {X 0.216,Y -581.473,Z 599.407,A 0.000,B 0.000,C 90.000,E1 109.214} C_DIS
LIN {X 0.108,Y -584.816,Z 599.402,A 0.000,B 0.000,C 90.000,E1 108.417} C_DIS
LIN {X 0.176,Y -586.890,Z 599.399,A 0.000,B 0.000,C 90.000,E1 107.873} C_DIS
LIN {X -0.065,Y -589.638,Z 599.395,A 0.000,B 0.000,C 90.000,E1 107.094} C_DIS
LIN {X 0.034,Y -591.480,Z 599.392,A 0.000,B 0.000,C 90.000,E1 106.551} C_DIS
LIN {X -0.200,Y -595.506,Z 599.385,A 0.000,B 0.000,C 90.000,E1 105.245} C_DIS
LIN {X -0.055,Y -602.020,Z 599.373,A 0.000,B 0.000,C 90.000,E1 103.119} C_DIS
LIN {X -0.196,Y -607.896,Z 599.363,A 0.000,B 0.000,C 90.000,E1 101.299} C_DIS
LIN {X -0.075,Y -612.807,Z 599.354,A 0.000,B 0.000,C 90.000,E1 99.726} C_DIS
LIN {X -0.314,Y -616.686,Z 599.347,A 0.000,B 0.000,C 90.000,E1 98.454} C_DIS
LIN {X 0.131,Y -620.309,Z 599.340,A 0.000,B 0.000,C 90.000,E1 97.125} C_DIS
LIN {X 0.019,Y -623.777,Z 599.333,A 0.000,B 0.000,C 90.000,E1 95.853} C_DIS
LIN {X -0.108,Y -626.708,Z 599.326,A 0.000,B 0.000,C 90.000,E1 94.588} C_DIS
LIN {X -0.297,Y -628.210,Z 599.321,A 0.000,B 0.000,C 90.000,E1 93.841} C_DIS
LIN {X -0.121,Y -630.028,Z 599.316,A 0.000,B 0.000,C 90.000,E1 92.808} C_DIS
LIN {X -0.192,Y -631.933,Z 599.309,A 0.000,B 0.000,C 90.000,E1 91.547} C_DIS
LIN {X -0.092,Y -632.595,Z 599.306,A 0.000,B 0.000,C 90.000,E1 91.031} C_DIS
LIN {X 0.127,Y -633.572,Z 599.300,A 0.000,B 0.000,C 90.000,E1 90.000} C_DIS
LIN {X -0.017,Y -634.053,Z 599.296,A 0.000,B 0.000,C 90.000,E1 89.255} C_DIS
LIN {X -0.159,Y -634.313,Z 599.292,A 0.000,B 0.000,C 90.000,E1 88.511} C_DIS
LIN {X -0.280,Y -634.378,Z 599.287,A 0.000,B 0.000,C 90.000,E1 87.764} C_DIS
LIN {X -0.017,Y -634.121,Z 599.282,A 0.000,B 0.000,C 90.000,E1 86.731} C_DIS
LIN {X 0.240,Y -633.531,Z 599.276,A 0.000,B 0.000,C 90.000,E1 85.698} C_DIS
LIN {X -0.149,Y -632.697,Z 599.271,A 0.000,B 0.000,C 90.000,E1 84.723} C_DIS
LIN {X 0.137,Y -631.682,Z 599.265,A 0.000,B 0.000,C 90.000,E1 83.685} C_DIS
LIN {X -0.218,Y -630.339,Z 599.259,A 0.000,B 0.000,C 90.000,E1 82.704} C_DIS
LIN {X 0.119,Y -628.605,Z 599.254,A 0.000,B 0.000,C 90.000,E1 81.659} C_DIS
LIN {X -0.281,Y -626.639,Z 599.248,A 0.000,B 0.000,C 90.000,E1 80.679} C_DIS
LIN {X 0.004,Y -624.494,Z 599.242,A 0.000,B 0.000,C 90.000,E1 79.634} C_DIS
LIN {X 0.159,Y -621.521,Z 599.235,A 0.000,B 0.000,C 90.000,E1 78.342} C_DIS
LIN {X -0.242,Y -618.981,Z 599.230,A 0.000,B 0.000,C 90.000,E1 77.353} C_DIS
LIN {X 0.052,Y -616.182,Z 599.224,A 0.000,B 0.000,C 90.000,E1 76.297} C_DIS
LIN {X 0.212,Y -612.422,Z 599.217,A 0.000,B 0.000,C 90.000,E1 74.991} C_DIS
LIN {X 0.228,Y -610.005,Z 599.212,A 0.000,B 0.000,C 90.000,E1 74.212} C_DIS
LIN {X 0.051,Y -607.389,Z 599.208,A 0.000,B 0.000,C 90.000,E1 73.449} C_DIS
LIN {X 0.015,Y -604.479,Z 599.204,A 0.000,B 0.000,C 90.000,E1 72.670} C_DIS
LIN {X 0.137,Y -601.286,Z 599.199,A 0.000,B 0.000,C 90.000,E1 71.873} C_DIS
LIN {X -0.008,Y -597.222,Z 599.194,A 0.000,B 0.000,C 90.000,E1 70.967} C_DIS
LIN {X -0.207,Y -592.767,Z 599.189,A 0.000,B 0.000,C 90.000,E1 70.061} C_DIS
LIN {X -0.197,Y -588.711,Z 599.185,A 0.000,B 0.000,C 90.000,E1 69.263} C_DIS
LIN {X -0.229,Y -584.247,Z 599.180,A 0.000,B 0.000,C 90.000,E1 68.465} C_DIS
LIN {X -0.103,Y -579.502,Z 599.176,A 0.000,B 0.000,C 90.000,E1 67.667} C_DIS
LIN {X 0.114,Y -575.186,Z 599.172,A 0.000,B 0.000,C 90.000,E1 66.997} C_DIS
LIN {X -0.283,Y -570.128,Z 599.169,A 0.000,B 0.000,C 90.000,E1 66.357} C_DIS
LIN {X -0.107,Y -565.738,Z 599.166,A 0.000,B 0.000,C 90.000,E1 65.793} C_DIS
LIN {X 0.037,Y -560.984,Z 599.162,A 0.000,B 0.000,C 90.000,E1 65.229} C_DIS
LIN {X 0.189,Y -555.852,Z 599.159,A 0.000,B 0.000,C 90.000,E1 64.665} C_DIS
LIN {X 0.057,Y -551.754,Z 599.157,A 0.000,B 0.000,C 90.000,E1 64.280} C_DIS
